METHOD M_Run
IF NOT _attached THEN
    RETURN;
END_IF
CASE _step OF
    0:  // initialize
        M_Step(StepNo := 0, StepName := 'project.step.pressAutoInitialize',
            Awaits := 0, AwaitingLabel := '', TimeClass := E_TimeClass.WORK, ExpectedTime := T#0S, Branch := 0);
        _outCmd.CycleCompleted := FALSE;
        _retVal := E_StepResult.ADVANCE;
        M_Advance(OnAdvance := 100, OnJump1 := -1, OnJump2 := -1, OnJump3 := -1 );
    100:  // await a fresh two-hand start (the §8.11.1 cycle-start marker)
        M_Step(StepNo := 100, StepName := 'project.step.pressAwaitTwoHand',
            Awaits := 0, AwaitingLabel := '', TimeClass := E_TimeClass.WAIT_OPERATOR, ExpectedTime := T#0S, Branch := 0);
        _outCmd.CycleCompleted := FALSE;
        _partReady := M_Await(Idx := 1, Label := 'project.condition.partPresent',
            Ok := _partPresentSensor.OutImm.Value AND _partPresentSensor.OutImm.Quality);
        _airReady := M_Await(Idx := 2, Label := 'project.condition.airPressureOk',
            Ok := _airPressureMonitor.OutImm.PressureOk);
        IF _stationCfg.RequireTwoHandStart THEN
            _startReady := M_Await(Idx := 3, Label := 'project.condition.twoHandStart', Ok := _startLatched);
        ELSE
            _startReady := TRUE;
        END_IF
        IF M_StopPending() THEN
            M_StopNow();                       // stop accepted BETWEEN cycles: no phantom cycle
        ELSIF _partReady AND _airReady AND _startReady THEN
            // §3.16.3 receive once per PHYSICAL part. The N180 two-hand abort returns
            // here with the same part still in the machine and nothing processed, so a
            // second M_PartReceived would open a duplicate record for one part.
            // M_PartStarted (N150) is deliberately NOT guarded: each pass is a genuine
            // processing attempt on that part.
            IF NOT _partInMachine THEN
                _traceAccepted := M_PartReceived();
                _partInMachine := TRUE;
            END_IF
            _retVal := E_StepResult.ADVANCE;
        END_IF
        M_Advance(OnAdvance := 110, OnJump1 := -1, OnJump2 := -1, OnJump3 := -1);
    110:  // ram up
        M_Step(StepNo := 110, StepName := 'project.step.pressRamUp',
            Awaits := _pressRam, AwaitingLabel := 'PressRam.RETRACT', TimeClass := E_TimeClass.WORK, ExpectedTime := T#0S, Branch := 0);
        IF M_TryIssue(Steppable := TRUE) THEN
            _pressRam.Abort := FALSE; _pressRam.Command := E_CylinderCommand.RETRACT; _pressRam.Execute := TRUE;
        END_IF
        IF _pressRam.Done THEN _pressRam.Execute := FALSE; _retVal := E_StepResult.ADVANCE; END_IF
        M_Advance(OnAdvance := 130, OnJump1 := -1, OnJump2 := -1, OnJump3 := -1);
    130:  // door open
        M_Step(StepNo := 130, StepName := 'project.step.pressDoorOpen',
            Awaits := _door, AwaitingLabel := 'Door.RETRACT', TimeClass := E_TimeClass.WORK, ExpectedTime := T#0S, Branch := 0);
        IF M_TryIssue(Steppable := TRUE) THEN
            _door.Abort := FALSE; _door.Command := E_CylinderCommand.RETRACT; _door.Execute := TRUE;
        END_IF
        IF _door.Done THEN _door.Execute := FALSE; _retVal := E_StepResult.ADVANCE; END_IF
        M_Advance(OnAdvance := 150, OnJump1 := -1, OnJump2 := -1, OnJump3 := -1);
    150:  // slide inside (value-adding sequence begins)
        M_Step(StepNo := 150, StepName := 'project.step.pressSlideInside',
            Awaits := _partSlide, AwaitingLabel := 'PartSlide.EXTEND', TimeClass := E_TimeClass.WORK, ExpectedTime := T#0S, Branch := 0);
        IF M_TryIssue(Steppable := TRUE) THEN
            M_PartStarted();
            _partSlide.Abort := FALSE; _partSlide.Command := E_CylinderCommand.EXTEND; _partSlide.Execute := TRUE;
        END_IF
        IF _partSlide.Done THEN _partSlide.Execute := FALSE; _retVal := E_StepResult.ADVANCE; END_IF
        M_Advance(OnAdvance := 170, OnJump1 := -1, OnJump2 := -1, OnJump3 := -1);
    170:  // transfer settle
        M_Step(StepNo := 170, StepName := 'project.step.pressTransferSettle',
            Awaits := 0, AwaitingLabel := '', TimeClass := E_TimeClass.WORK, ExpectedTime := _parCfg.TransferSettleTime, Branch := 0);
        _retVal := M_Delay(PT := _parCfg.TransferSettleTime);
        M_Advance(OnAdvance := 180, OnJump1 := -1, OnJump2 := -1, OnJump3 := -1);
    180:  // door close. Releasing a two-hand button while the door is moving is an
          // operator abort, not a fault: the door goes back up, the part slides out,
          // and the cycle returns to the two-hand wait (§6.10 jump). Completion wins
          // if the door finished in the same scan the button was released.
        M_Step(StepNo := 180, StepName := 'project.step.pressDoorClose',
            Awaits := _door, AwaitingLabel := 'Door.EXTEND', TimeClass := E_TimeClass.WORK, ExpectedTime := T#0S, Branch := 0);
        _twoHandHeldDuringClose := M_Await(Idx := 1,
            Label := 'project.condition.twoHandHeldDuringDoorClose',
            Ok := _twoHand.OutImm.SafeActive OR NOT _stationCfg.RequireTwoHandStart);
        IF M_TryIssue(Steppable := TRUE) THEN
            _door.Abort := FALSE; _door.Command := E_CylinderCommand.EXTEND; _door.Execute := TRUE;
        END_IF
        IF _door.Done THEN
            _door.Execute := FALSE;
            _retVal := E_StepResult.ADVANCE;
        ELSIF NOT _twoHandHeldDuringClose THEN
            _door.Execute := FALSE;             // §6.1 Execute-drop reset releases the close
            // §6.9(e) — a WARNING, not a fault: the release is designed operator
            // behaviour and the chain already owns the recovery below, so nothing
            // stops. It is recorded because a cycle was abandoned with the part
            // still in the machine, and the §3.13 chart marks this step for it.
            // The base raises it once per visit however many scans this runs.
            _closeAbortWarned := M_RaiseWarning(
                Reason := PL_PressReasons.PRESS_TWO_HAND_RELEASED,
                DescriptionKey := 'project.warning.twoHandReleasedDuringDoorClose',
                Severity := E_Severity.LOW, Category := E_Category.PROCESS);
            _retVal := E_StepResult.JUMP1;      // released -> reopen and clear the part
        END_IF
        M_Advance(OnAdvance := 200, OnJump1 := 185, OnJump2 := -1, OnJump3 := -1);
    185:  // two-hand released during closing: take the door back up
        M_Step(StepNo := 185, StepName := 'project.step.pressDoorReopen',
            Awaits := _door, AwaitingLabel := 'Door.RETRACT', TimeClass := E_TimeClass.WORK, ExpectedTime := T#0S, Branch := 0);
        IF M_TryIssue(Steppable := TRUE) THEN
            _door.Abort := FALSE; _door.Command := E_CylinderCommand.RETRACT; _door.Execute := TRUE;
        END_IF
        IF _door.Done THEN _door.Execute := FALSE; _retVal := E_StepResult.ADVANCE; END_IF
        M_Advance(OnAdvance := 190, OnJump1 := -1, OnJump2 := -1, OnJump3 := -1);
    190:  // slide the part back out, then return to the two-hand wait. The start latch
          // is dropped so the cycle cannot resume without a fresh two-hand press.
        M_Step(StepNo := 190, StepName := 'project.step.pressSlideOutsideAfterAbort',
            Awaits := _partSlide, AwaitingLabel := 'PartSlide.RETRACT', TimeClass := E_TimeClass.WORK, ExpectedTime := T#0S, Branch := 0);
        IF M_TryIssue(Steppable := TRUE) THEN
            _partSlide.Abort := FALSE; _partSlide.Command := E_CylinderCommand.RETRACT; _partSlide.Execute := TRUE;
        END_IF
        IF _partSlide.Done THEN
            _partSlide.Execute := FALSE;
            _startLatched := FALSE;
            _retVal := E_StepResult.ADVANCE;
        END_IF
        M_Advance(OnAdvance := 100, OnJump1 := -1, OnJump2 := -1, OnJump3 := -1);
    200:  // ram down. THIS step owns the not-reached disposition, so it does NOT hand
          // the ram to the §6.9 auto-rollup: an awaited child fault is adopted by the
          // Unit (ERROR, _step := 0) before _M_Dispatch runs, and the chain would stop
          // before it could ask the operator anything. The wait is still named (§6.9(b))
          // and the cylinder still raises its own CYL_NOT_EXTENDED alarm.
        M_Step(StepNo := 200, StepName := 'project.step.pressRamDown',
            Awaits := 0, AwaitingLabel := '', TimeClass := E_TimeClass.WORK, ExpectedTime := T#0S, Branch := 0);
        _ramReached := M_Await(Idx := 1, Label := 'project.condition.pressRamExtended',
            Ok := _pressRam.Done);
        IF M_TryIssue(Steppable := TRUE) THEN
            _pressRam.Abort := FALSE; _pressRam.Command := E_CylinderCommand.EXTEND; _pressRam.Execute := TRUE;
        END_IF
        IF _pressRam.Done THEN
            _pressRam.Execute := FALSE;
            _retVal := E_StepResult.ADVANCE;
        ELSIF _pressRam.Error THEN
            // §6.9(e) — publish the ram's own first-out (CYL_NOT_EXTENDED, with its
            // text and IO tag) on the Unit and on this row of the §3.13 chart, and
            // do NOT adopt it: the confirmation + scrap below IS the handling, so a
            // fault here would replace a designed recovery. Saying nothing is what
            // left the failure visible only on the ram itself.
            _ramFailureReported := M_ReportFromChild(Source := _pressRam);
            _pressRam.Execute := FALSE;         // §6.1 Execute-drop reset returns the ram to READY
            _retVal := E_StepResult.JUMP1;      // did not reach -> operator confirmation
        END_IF
        M_Advance(OnAdvance := 220, OnJump1 := 210, OnJump2 := -1, OnJump3 := -1);
    210:  // press did not reach: the operator confirms the failure before the part is
          // scrapped. A scrap is deliberate, so there is no timeout default (§6.11).
        M_Step(StepNo := 210, StepName := 'project.step.pressNotReachedConfirm',
            Awaits := 0, AwaitingLabel := '', TimeClass := E_TimeClass.WAIT_OPERATOR, ExpectedTime := T#0S, Branch := 0);
        _decisionRequest.Prompt := 'project.decision.pressNotReached';
        _decisionRequest.Options[1] := 'project.decision.confirmScrapAndReturn';
        _decisionRequest.Default := 0;
        _decisionRequest.Timeout := T#0S;
        M_AskDecision(Req := _decisionRequest);
        _answer := M_TakeDecision();
        IF _answer = 1 THEN
            _retVal := E_StepResult.ADVANCE;
        ELSE
            _failureConfirmed := M_Await(Idx := 1,
                Label := 'project.condition.pressFailureConfirmation', Ok := FALSE);
        END_IF
        M_Advance(OnAdvance := 215, OnJump1 := -1, OnJump2 := -1, OnJump3 := -1);
    215:  // disposition the part NOK, then rejoin the shared return-to-start step
        M_Step(StepNo := 215, StepName := 'project.step.pressScrapPart',
            Awaits := 0, AwaitingLabel := '', TimeClass := E_TimeClass.WORK, ExpectedTime := T#0S, Branch := 0);
        _partProcessed := M_PartProcessed(Verdict := E_Verdict.NOK,
            Reason := PL_ModuleReasons.CYL_NOT_EXTENDED);
        _partDispositioned := TRUE;             // N999 must not also count it good
        _partInMachine := FALSE;                // dispositioned: the next one is a new part
        _outCmd.CycleCompleted := FALSE;
        _retVal := E_StepResult.ADVANCE;
        M_Advance(OnAdvance := 240, OnJump1 := -1, OnJump2 := -1, OnJump3 := -1);
    220:  // press dwell — two-hand must stay held; releasing it HOLDS the dwell
        M_Step(StepNo := 220, StepName := 'project.step.pressDwell',
            Awaits := 0, AwaitingLabel := '', TimeClass := E_TimeClass.WORK, ExpectedTime := _parCfg.PressSettleTime, Branch := 0);
        // Releasing the button mid-dwell is the designed way to stop pressing, so it
        // is a named wait (§6.9(b)), not a fault: the ram's outputs come off, the
        // dwell timer freezes where it is because M_Delay is not called, and pressing
        // again restores the force and finishes the remaining dwell. Faulting here
        // charged an unrecoverable downtime event for normal operator behaviour.
        _dwellTwoHandHeld := M_Await(Idx := 1, Label := 'project.condition.twoHandHeldDuringPress',
            Ok := _twoHand.OutImm.SafeActive OR NOT _stationCfg.RequireTwoHandStart);
        IF NOT _dwellTwoHandHeld THEN
            _pressRam.WithdrawOutputs();
        ELSE
            // The press force is the valve latched by the EXTEND that step 200 already
            // completed, so after a withdraw only this call re-energizes it — and the
            // ram re-checks its own extend permit before it does (§7.2).
            _pressRam.RestoreOutputs();
            _retVal := M_Delay(PT := _parCfg.PressSettleTime);
        END_IF
        M_Advance(OnAdvance := 230, OnJump1 := -1, OnJump2 := -1, OnJump3 := -1);
    230:  // record the applied dwell (§3.16.1 measured value)
        M_Step(StepNo := 230, StepName := 'project.step.pressRecordResult',
            Awaits := 0, AwaitingLabel := '', TimeClass := E_TimeClass.WORK, ExpectedTime := T#0S, Branch := 0);
        _recordAccepted := M_PartRecord(RecordName := 'PressDwell',
            Value := DINT_TO_LREAL(TIME_TO_DINT(_parCfg.PressSettleTime)),
            Minimum := 0, Maximum := 30000,
            Target := DINT_TO_LREAL(TIME_TO_DINT(_parCfg.PressSettleTime)), EngUnit := 'ms');
        _retVal := E_StepResult.ADVANCE;
        M_Advance(OnAdvance := 240, OnJump1 := -1, OnJump2 := -1, OnJump3 := -1);
    240:  // return to the shared load-safe position (composite step)
        _retVal := M_RunSub(Chain := _loadPosition, BaseStepNo := 240);
        M_Advance(OnAdvance := 999, OnJump1 := -1, OnJump2 := -1, OnJump3 := -1);
    999:  // cycle complete — write result, count by verdict, loop (§8.11.1 finish marker)
        M_Step(StepNo := 999, StepName := 'project.step.pressAutoComplete',
            Awaits := 0, AwaitingLabel := '', TimeClass := E_TimeClass.WORK, ExpectedTime := T#0S, Branch := 0);
        _outCmd.CycleCompleted := TRUE;
        IF _partDispositioned THEN
            _partDispositioned := FALSE;       // N260 already set the NOK verdict
        ELSE
            _partProcessed := M_PartProcessed(Verdict := E_Verdict.OK, Reason := E_Reason.NONE);
            IF NOT _partProcessed THEN
                M_CountGood();                 // §3.9: no carrier configured — count directly
            END_IF
        END_IF
        _partInMachine := FALSE;               // processed: the next one is a new part
        _startLatched := FALSE;
        IF M_EndOfCycle() THEN
            _retVal := E_StepResult.ADVANCE;   // stop NOT requested: loop to N100
        END_IF
        M_Advance(OnAdvance := 100, OnJump1 := -1, OnJump2 := -1, OnJump3 := -1);
ELSE
    M_Fault(Reason := E_Reason.STEP_STALLED, DescriptionKey := 'std.error.undefinedStep');
END_CASE
END_METHOD

METHOD Setup : BOOL
VAR_INPUT
    Host : I_SequenceHost;
END_VAR
VAR_IN_OUT
    PressRam : FB_CylinderCM;
    Door : FB_CylinderCM;
    PartSlide : FB_CylinderCM;
    TwoHand : FB_TwoHandStartCM;
    PartPresentSensor : FB_DigitalInputCM;
    AirPressureMonitor : FB_AirPressureMonitorCM;
    ParCfg : ST_PneumaticPressParCfg;
    StationCfg : ST_PneumaticPressStationCfg;
    OutCmd : ST_PneumaticPressOutCmd;
    StartLatched : BOOL;
END_VAR
_pressRam REF= PressRam;
_door REF= Door;
_partSlide REF= PartSlide;
_twoHand REF= TwoHand;
_partPresentSensor REF= PartPresentSensor;
_airPressureMonitor REF= AirPressureMonitor;
_parCfg REF= ParCfg;
_stationCfg REF= StationCfg;
_outCmd REF= OutCmd;
_startLatched REF= StartLatched;
Setup := M_Attach(Host := Host) AND __ISVALIDREF(_pressRam) AND __ISVALIDREF(_door)
    AND __ISVALIDREF(_partSlide) AND __ISVALIDREF(_twoHand)
    AND __ISVALIDREF(_partPresentSensor) AND __ISVALIDREF(_airPressureMonitor)
    AND __ISVALIDREF(_parCfg) AND __ISVALIDREF(_outCmd) AND __ISVALIDREF(_startLatched)
    AND _loadPosition.Setup(Host := Host, PressRam := PressRam, Door := Door, PartSlide := PartSlide);
END_METHOD

END_FUNCTION_BLOCK

// ---- Fraktal_Press_Demo/01_PneumaticPress/Sequences/FB_SFC_PressDemoAuto.TcPOU
// SFC rendition of FB_PressDemoAuto - identical behaviour, chart-language
// transitions. Every step action below sets the shared `_retVal`; the chart's
// transitions read it, and the owner calls M_BeginScan() once per PLC cycle
// before executing this chart so the result cannot survive into the next scan
// (Core §6.8). The ST twin remains FB_PressDemoAuto; keep the two in step.
FUNCTION_BLOCK INTERNAL FB_SFC_PressDemoAuto EXTENDS FB_SequenceBase
VAR
    _partReady, _airReady, _startReady : BOOL;
    _dwellTwoHandHeld : BOOL;          // N220 named wait: two-hand held through the dwell
    _decisionRequest : ST_DecisionRequest;   // §6.11 not-reached confirmation
    _answer : INT;
    _ramReached, _failureConfirmed : BOOL;   // N200/N210 named waits
    _twoHandHeldDuringClose : BOOL;
    _closeAbortWarned : BOOL;                // N180 §6.9(e) message result
    _ramFailureReported : BOOL;              // N200 §6.9(e) message result          // N180 named wait
    _partInMachine : BOOL;                   // §3.16.3 the part is already received
    _partDispositioned : BOOL;               // N260 already set the verdict
    _traceAccepted, _recordAccepted, _partProcessed : BOOL;
    {attribute 'OPC.UA.DA' := '0'}
    _pressRam : REFERENCE TO FB_CylinderCM;
    {attribute 'OPC.UA.DA' := '0'}
    _door : REFERENCE TO FB_CylinderCM;
    {attribute 'OPC.UA.DA' := '0'}
    _partSlide : REFERENCE TO FB_CylinderCM;
    {attribute 'OPC.UA.DA' := '0'}
    _twoHand : REFERENCE TO FB_TwoHandStartCM;
    {attribute 'OPC.UA.DA' := '0'}
    _partPresentSensor : REFERENCE TO FB_DigitalInputCM;
    {attribute 'OPC.UA.DA' := '0'}
    _airPressureMonitor : REFERENCE TO FB_AirPressureMonitorCM;
    {attribute 'OPC.UA.DA' := '0'}
    _parCfg : REFERENCE TO ST_PneumaticPressParCfg;
    // §3.8a - the CELL's own policy, held separately from the MODEL's data and
    // referenced exactly like _parCfg, so each step reads whichever structure
    // actually owns the value it is asking about.
    {attribute 'OPC.UA.DA' := '0'}
    _stationCfg : REFERENCE TO ST_PneumaticPressStationCfg;
    {attribute 'OPC.UA.DA' := '0'}
    _outCmd : REFERENCE TO ST_PneumaticPressOutCmd;
    {attribute 'OPC.UA.DA' := '0'}
    _startLatched : REFERENCE TO BOOL;
    {attribute 'OPC.UA.DA' := '0'}
    _loadPosition : FB_PressDemoLoadPosition;
END_VAR

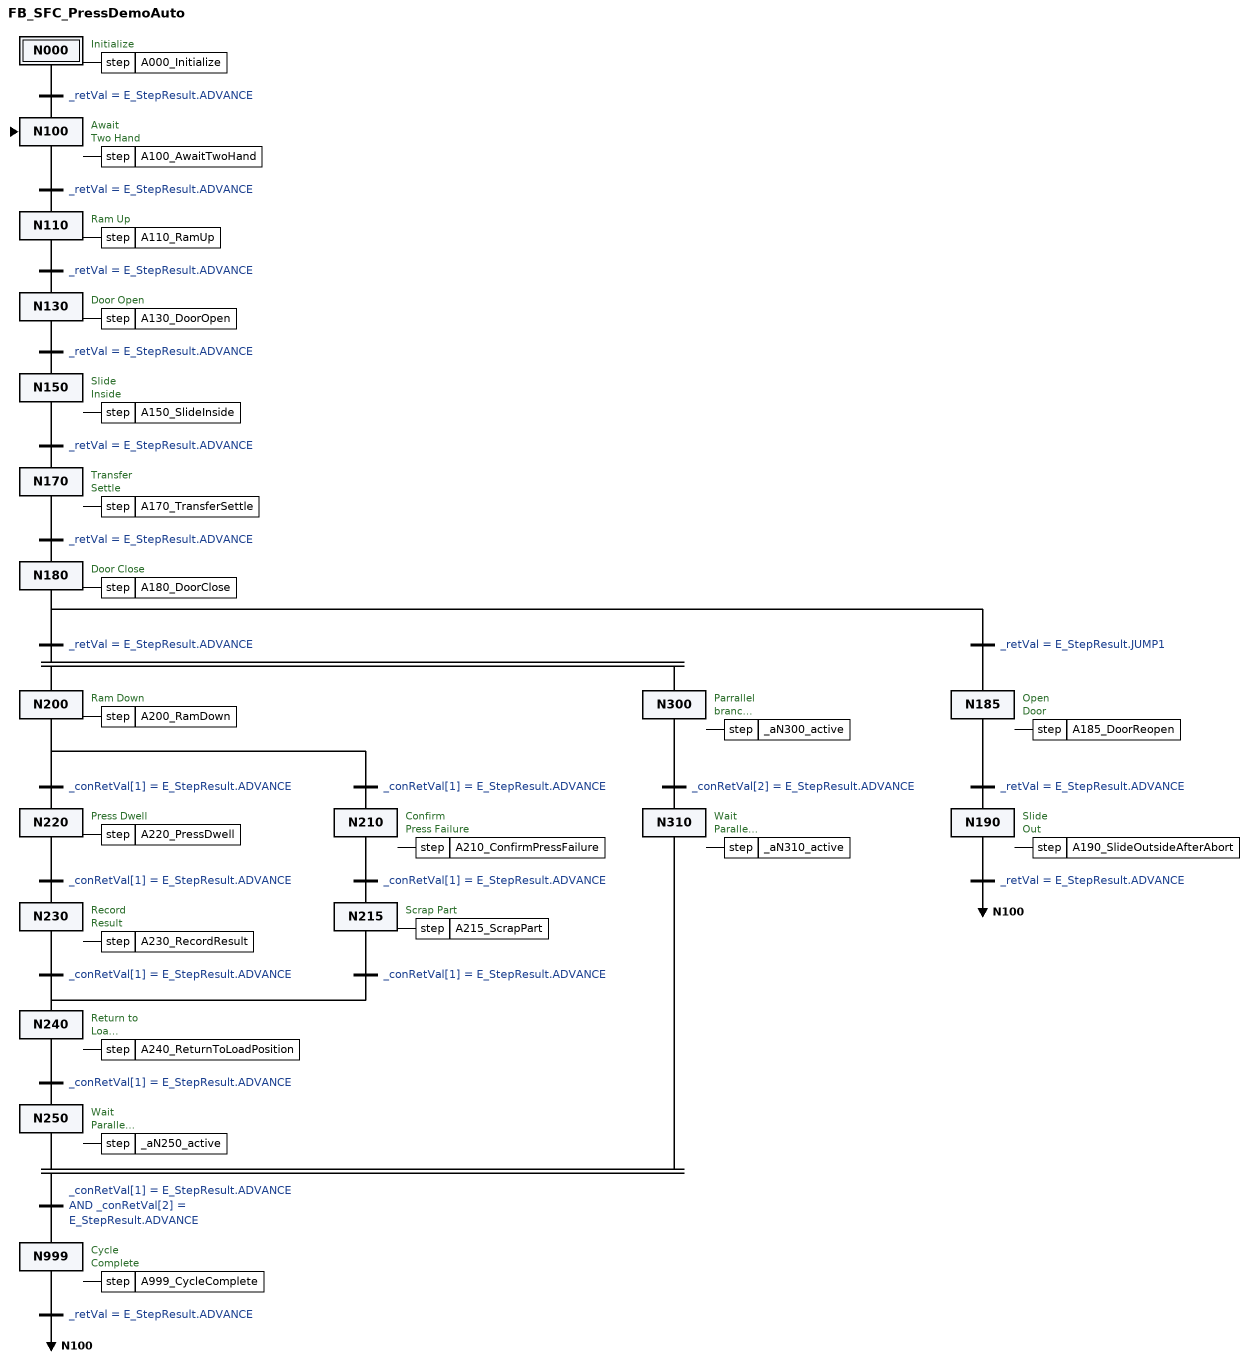
// Initialize
INITIAL_STEP N000:
    A000_Initialize(N);  // step action
END_STEP
TRANSITION FROM N000 TO N100
    := _retVal = E_StepResult.ADVANCE;
END_TRANSITION
// Await
// Two Hand
STEP N100:
    A100_AwaitTwoHand(N);  // step action
END_STEP
TRANSITION FROM N100 TO N110
    := _retVal = E_StepResult.ADVANCE;
END_TRANSITION
// Ram Up
STEP N110:
    A110_RamUp(N);  // step action
END_STEP
TRANSITION FROM N110 TO N130
    := _retVal = E_StepResult.ADVANCE;
END_TRANSITION
// Door Open
STEP N130:
    A130_DoorOpen(N);  // step action
END_STEP
TRANSITION FROM N130 TO N150
    := _retVal = E_StepResult.ADVANCE;
END_TRANSITION
// Slide
// Inside
STEP N150:
    A150_SlideInside(N);  // step action
END_STEP
TRANSITION FROM N150 TO N170
    := _retVal = E_StepResult.ADVANCE;
END_TRANSITION
// Transfer
// Settle
STEP N170:
    A170_TransferSettle(N);  // step action
END_STEP
TRANSITION FROM N170 TO N180
    := _retVal = E_StepResult.ADVANCE;
END_TRANSITION
// Door Close
STEP N180:
    A180_DoorClose(N);  // step action
END_STEP
TRANSITION FROM N180 TO (N200, N300)
    := _retVal = E_StepResult.ADVANCE;
END_TRANSITION
// Ram Down
STEP N200:
    A200_RamDown(N);  // step action
END_STEP
TRANSITION FROM N200 TO N220
    := _conRetVal[1] = E_StepResult.ADVANCE;
END_TRANSITION
// Press Dwell
STEP N220:
    A220_PressDwell(N);  // step action
END_STEP
TRANSITION FROM N220 TO N230
    := _conRetVal[1] = E_StepResult.ADVANCE;
END_TRANSITION
// Record
// Result
STEP N230:
    A230_RecordResult(N);  // step action
END_STEP
TRANSITION FROM N230 TO N240
    := _conRetVal[1] = E_StepResult.ADVANCE;
END_TRANSITION
TRANSITION FROM N200 TO N210
    := _conRetVal[1] = E_StepResult.ADVANCE;
END_TRANSITION
// Confirm
// Press Failure
STEP N210:
    A210_ConfirmPressFailure(N);  // step action
END_STEP
TRANSITION FROM N210 TO N215
    := _conRetVal[1] = E_StepResult.ADVANCE;
END_TRANSITION
// Scrap Part
STEP N215:
    A215_ScrapPart(N);  // step action
END_STEP
TRANSITION FROM N215 TO N240
    := _conRetVal[1] = E_StepResult.ADVANCE;
END_TRANSITION
// Return to
// Load
// Position
STEP N240:
    A240_ReturnToLoadPosition(N);  // step action
END_STEP
TRANSITION FROM N240 TO N250
    := _conRetVal[1] = E_StepResult.ADVANCE;
END_TRANSITION
// Wait
// Parallel
// Branch
STEP N250:
    _aN250_active(N);  // step action
END_STEP
// Parrallel
// branch
// example
STEP N300:
    _aN300_active(N);  // step action
END_STEP
TRANSITION FROM N300 TO N310
    := _conRetVal[2] = E_StepResult.ADVANCE;
END_TRANSITION
// Wait
// Parallel
// Branch
STEP N310:
    _aN310_active(N);  // step action
END_STEP
TRANSITION FROM N180 TO N185
    := _retVal = E_StepResult.JUMP1;
END_TRANSITION
// Open
// Door
STEP N185:
    A185_DoorReopen(N);  // step action
END_STEP
TRANSITION FROM N185 TO N190
    := _retVal = E_StepResult.ADVANCE;
END_TRANSITION
// Slide
// Out
STEP N190:
    A190_SlideOutsideAfterAbort(N);  // step action
END_STEP
TRANSITION FROM N190 TO N100
    := _retVal = E_StepResult.ADVANCE;
END_TRANSITION
TRANSITION FROM (N250, N310) TO N999
    := _conRetVal[1] = E_StepResult.ADVANCE AND _conRetVal[2] = E_StepResult.ADVANCE;
END_TRANSITION
// Cycle
// Complete
STEP N999:
    A999_CycleComplete(N);  // step action
END_STEP
TRANSITION FROM N999 TO N100
    := _retVal = E_StepResult.ADVANCE;
END_TRANSITION

ACTION _aN250_active:
// N250 — leg 1 waits at the join. §6.12: the parallel divergence after A180 is
// drawn INSIDE this POU, so both legs share the FB and each leg step says which leg
// it is through `Branch` on its own step record - a leg can never be declared
// without recording a step.
//
// NEITHER leg is the main line. A simultaneous divergence has N equal legs, so
// numbering one of them 0 would have made it look subordinate on the §3.13 chart
// and left `_retVal` meaning two different things depending on where you were
// reading it. `_retVal` is the single-threaded line before and after the fork;
// inside it, leg 1 is `_conRetVal[1]` and leg 2 is `_conRetVal[2]`.
M_Step(StepNo := 250, StepName := 'project.step.pressAwaitParallelBranch', Awaits := 0,
    AwaitingLabel := '', TimeClass := E_TimeClass.WORK, ExpectedTime := T#0S,
    Branch := 1);
_conRetVal[1] := E_StepResult.ADVANCE;
END_ACTION

ACTION _aN300_active:
// N300 — concurrent leg 1, first step. Everything a normal step does is available
// here; `Branch := 1` is what keeps this leg's issue latch, delay and message
// separate from the main line's, so both legs can command their own children in
// the same scan. This example commands nothing: the press has one work position,
// and inventing a second would change what the machine does. A real one goes here.
M_Step(StepNo := 300, StepName := 'project.step.pressParallelWork', Awaits := 0,
    AwaitingLabel := '', TimeClass := E_TimeClass.WORK, ExpectedTime := T#0S,
    Branch := 2);
_conRetVal[2] := E_StepResult.ADVANCE;   // leg 2's result; leg 1 uses _conRetVal[1]
END_ACTION

ACTION _aN310_active:
// N310 — concurrent leg 1 waits at the join. A parallel divergence joins only when
// EVERY leg has reached its last step, so each leg needs a terminal step to sit in
// while the others finish; this is that step for leg 1, and A250 is the main
// line's.
M_Step(StepNo := 310, StepName := 'project.step.pressAwaitParallelJoin', Awaits := 0,
    AwaitingLabel := '', TimeClass := E_TimeClass.WORK, ExpectedTime := T#0S,
    Branch := 2);
_conRetVal[2] := E_StepResult.ADVANCE;
END_ACTION

ACTION A000_Initialize:
// N000 step action. SFC step `A000_Initialize` calls this; its transition reads
// `_retVal = E_StepResult.ADVANCE`. Body is the ST chart's branch verbatim,
// without M_Advance - the chart runtime owns the transition.
M_Step(StepNo := 0, StepName := 'project.step.pressAutoInitialize',
    Awaits := 0, AwaitingLabel := '', TimeClass := E_TimeClass.WORK, ExpectedTime := T#0S, Branch := 0);
_outCmd.CycleCompleted := FALSE;
_retVal := E_StepResult.ADVANCE;
END_ACTION

ACTION A100_AwaitTwoHand:
// N100 step action. The §8.11.1 cycle-start marker; also the target of the
// N190 two-hand abort, which returns here with the same part still in place.
M_Step(StepNo := 100, StepName := 'project.step.pressAwaitTwoHand',
    Awaits := 0, AwaitingLabel := '', TimeClass := E_TimeClass.WAIT_OPERATOR, ExpectedTime := T#0S, Branch := 0);
_outCmd.CycleCompleted := FALSE;
_partReady := M_Await(Idx := 1, Label := 'project.condition.partPresent',
    Ok := _partPresentSensor.OutImm.Value AND _partPresentSensor.OutImm.Quality);
_airReady := M_Await(Idx := 2, Label := 'project.condition.airPressureOk',
    Ok := _airPressureMonitor.OutImm.PressureOk);
IF _stationCfg.RequireTwoHandStart THEN
    _startReady := M_Await(Idx := 3, Label := 'project.condition.twoHandStart', Ok := _startLatched);
ELSE
    _startReady := TRUE;
END_IF
IF M_StopPending() THEN
    M_StopNow();                       // stop accepted BETWEEN cycles: no phantom cycle
ELSIF _partReady AND _airReady AND _startReady THEN
    // §3.16.3 receive once per PHYSICAL part. The N180 two-hand abort returns
    // here with the same part still in the machine and nothing processed, so a
    // second M_PartReceived would open a duplicate record for one part.
    // M_PartStarted (N150) is deliberately NOT guarded: each pass is a genuine
    // processing attempt on that part.
    IF NOT _partInMachine THEN
        _traceAccepted := M_PartReceived();
        _partInMachine := TRUE;
    END_IF
    _retVal := E_StepResult.ADVANCE;
END_IF
END_ACTION

ACTION A110_RamUp:
// N110 step action. SFC step `A110_RamUp` calls this; its transition reads
// `_retVal = E_StepResult.ADVANCE`. Body is the ST chart's branch verbatim,
// without M_Advance - the chart runtime owns the transition.
M_Step(StepNo := 110, StepName := 'project.step.pressRamUp',
    Awaits := _pressRam, AwaitingLabel := 'PressRam.RETRACT', TimeClass := E_TimeClass.WORK, ExpectedTime := T#0S, Branch := 0);
IF M_TryIssue(Steppable := TRUE) THEN
    _pressRam.Abort := FALSE; _pressRam.Command := E_CylinderCommand.RETRACT; _pressRam.Execute := TRUE;
END_IF
IF _pressRam.Done THEN _pressRam.Execute := FALSE; _retVal := E_StepResult.ADVANCE; END_IF
END_ACTION

ACTION A130_DoorOpen:
// N130 step action. SFC step `A130_DoorOpen` calls this; its transition reads
// `_retVal = E_StepResult.ADVANCE`. Body is the ST chart's branch verbatim,
// without M_Advance - the chart runtime owns the transition.
M_Step(StepNo := 130, StepName := 'project.step.pressDoorOpen',
    Awaits := _door, AwaitingLabel := 'Door.RETRACT', TimeClass := E_TimeClass.WORK, ExpectedTime := T#0S, Branch := 0);
IF M_TryIssue(Steppable := TRUE) THEN
    _door.Abort := FALSE; _door.Command := E_CylinderCommand.RETRACT; _door.Execute := TRUE;
END_IF
IF _door.Done THEN _door.Execute := FALSE; _retVal := E_StepResult.ADVANCE; END_IF
END_ACTION

ACTION A150_SlideInside:
// N150 step action. SFC step `A150_SlideInside` calls this; its transition reads
// `_retVal = E_StepResult.ADVANCE`. Body is the ST chart's branch verbatim,
// without M_Advance - the chart runtime owns the transition.
M_Step(StepNo := 150, StepName := 'project.step.pressSlideInside',
    Awaits := _partSlide, AwaitingLabel := 'PartSlide.EXTEND', TimeClass := E_TimeClass.WORK, ExpectedTime := T#0S, Branch := 0);
IF M_TryIssue(Steppable := TRUE) THEN
    M_PartStarted();
    _partSlide.Abort := FALSE; _partSlide.Command := E_CylinderCommand.EXTEND; _partSlide.Execute := TRUE;
END_IF
IF _partSlide.Done THEN _partSlide.Execute := FALSE; _retVal := E_StepResult.ADVANCE; END_IF
END_ACTION

ACTION A170_TransferSettle:
// N170 step action. SFC step `A170_TransferSettle` calls this; its transition reads
// `_retVal = E_StepResult.ADVANCE`. Body is the ST chart's branch verbatim,
// without M_Advance - the chart runtime owns the transition.
M_Step(StepNo := 170, StepName := 'project.step.pressTransferSettle',
    Awaits := 0, AwaitingLabel := '', TimeClass := E_TimeClass.WORK, ExpectedTime := _parCfg.TransferSettleTime, Branch := 0);
_retVal := M_Delay(PT := _parCfg.TransferSettleTime);
END_ACTION

ACTION A180_DoorClose:
// N180 step action. Transition `_retVal = E_StepResult.ADVANCE` -> A200;
// the JUMP1 branch (`_retVal = E_StepResult.JUMP1`) -> A185.
//
// Releasing a two-hand button while the door is moving is an operator abort, not
// a fault: the door goes back up, the part slides out, and the cycle returns to
// the two-hand wait. Completion wins if the door finished in the same scan the
// button was released.
M_Step(StepNo := 180, StepName := 'project.step.pressDoorClose',
    Awaits := _door, AwaitingLabel := 'Door.EXTEND', TimeClass := E_TimeClass.WORK, ExpectedTime := T#0S, Branch := 0);
_twoHandHeldDuringClose := M_Await(Idx := 1,
    Label := 'project.condition.twoHandHeldDuringDoorClose',
    Ok := _twoHand.OutImm.SafeActive OR NOT _stationCfg.RequireTwoHandStart);
IF M_TryIssue(Steppable := TRUE) THEN
    _door.Abort := FALSE; _door.Command := E_CylinderCommand.EXTEND; _door.Execute := TRUE;
END_IF
IF _door.Done THEN
    _door.Execute := FALSE;
    _retVal := E_StepResult.ADVANCE;
ELSIF NOT _twoHandHeldDuringClose THEN
    _door.Execute := FALSE;             // §6.1 Execute-drop reset releases the close
    // §6.9(e) — a WARNING, not a fault: nothing stops, the JUMP1 branch below is
    // the recovery. Recorded because a cycle was abandoned with the part still in
    // the machine. Raised once per visit however many scans this action runs.
    _closeAbortWarned := M_RaiseWarning(
        Reason := PL_PressReasons.PRESS_TWO_HAND_RELEASED,
        DescriptionKey := 'project.warning.twoHandReleasedDuringDoorClose',
        Severity := E_Severity.LOW, Category := E_Category.PROCESS);
    _retVal := E_StepResult.JUMP1;      // released -> reopen and clear the part
END_IF
END_ACTION

ACTION A185_DoorReopen:
// N185 step action. Reached from A180 by JUMP1 when a two-hand button is
// released while the door closes. Advances to A190.
M_Step(StepNo := 185, StepName := 'project.step.pressDoorReopen',
    Awaits := _door, AwaitingLabel := 'Door.RETRACT', TimeClass := E_TimeClass.WORK, ExpectedTime := T#0S, Branch := 0);
IF M_TryIssue(Steppable := TRUE) THEN
    _door.Abort := FALSE; _door.Command := E_CylinderCommand.RETRACT; _door.Execute := TRUE;
END_IF
IF _door.Done THEN _door.Execute := FALSE; _retVal := E_StepResult.ADVANCE; END_IF
END_ACTION

ACTION A190_SlideOutsideAfterAbort:
// N190 step action. Slides the part out and drops the start latch, then its
// transition jumps back to A100, the two-hand wait. The start latch is dropped
// so the cycle cannot resume without a fresh two-hand press.
M_Step(StepNo := 190, StepName := 'project.step.pressSlideOutsideAfterAbort',
    Awaits := _partSlide, AwaitingLabel := 'PartSlide.RETRACT', TimeClass := E_TimeClass.WORK, ExpectedTime := T#0S, Branch := 0);
IF M_TryIssue(Steppable := TRUE) THEN
    _partSlide.Abort := FALSE; _partSlide.Command := E_CylinderCommand.RETRACT; _partSlide.Execute := TRUE;
END_IF
IF _partSlide.Done THEN
    _partSlide.Execute := FALSE;
    _startLatched := FALSE;
    _retVal := E_StepResult.ADVANCE;
END_IF
END_ACTION

ACTION A200_RamDown:
// N200 step action. Transition `_retVal = E_StepResult.ADVANCE` -> A220;
// the JUMP1 branch (`_retVal = E_StepResult.JUMP1`) -> A210.
// the ram to the §6.9 auto-rollup: an awaited child fault is adopted by the
// Unit (ERROR, _step := 0) before _M_Dispatch runs, and the chain would stop
// before it could ask the operator anything. The wait is still named (§6.9(b))
// and the cylinder still raises its own CYL_NOT_EXTENDED alarm.
M_Step(StepNo := 200, StepName := 'project.step.pressRamDown',
    Awaits := 0, AwaitingLabel := '', TimeClass := E_TimeClass.WORK, ExpectedTime := T#0S,
    Branch := 1);
_ramReached := M_Await(Idx := 1, Label := 'project.condition.pressRamExtended',
    Ok := _pressRam.Done);
IF M_TryIssue(Steppable := TRUE) THEN
    _pressRam.Abort := FALSE; _pressRam.Command := E_CylinderCommand.EXTEND; _pressRam.Execute := TRUE;
END_IF
IF _pressRam.Done THEN
    _pressRam.Execute := FALSE;
    _conRetVal[1] := E_StepResult.ADVANCE;
ELSIF _pressRam.Error THEN
    // §6.9(e) — publish the ram's own first-out on the Unit and on this row of the
    // §3.13 chart without adopting it: the confirmation + scrap below IS the
    // handling, so a fault here would replace a designed recovery.
    _ramFailureReported := M_ReportFromChild(Source := _pressRam);
    _pressRam.Execute := FALSE;         // §6.1 Execute-drop reset returns the ram to READY
    _conRetVal[1] := E_StepResult.JUMP1;      // did not reach -> operator confirmation
END_IF
END_ACTION

ACTION A210_ConfirmPressFailure:
// N210 step action. Reached from A200 by JUMP1; advances to A215.
// scrapped. A scrap is deliberate, so there is no timeout default (§6.11).
M_Step(StepNo := 210, StepName := 'project.step.pressNotReachedConfirm',
    Awaits := 0, AwaitingLabel := '', TimeClass := E_TimeClass.WAIT_OPERATOR, ExpectedTime := T#0S,
    Branch := 1);
_decisionRequest.Prompt := 'project.decision.pressNotReached';
_decisionRequest.Options[1] := 'project.decision.confirmScrapAndReturn';
_decisionRequest.Default := 0;
_decisionRequest.Timeout := T#0S;
M_AskDecision(Req := _decisionRequest);
_answer := M_TakeDecision();
IF _answer = 1 THEN
    _conRetVal[1] := E_StepResult.ADVANCE;
ELSE
    _failureConfirmed := M_Await(Idx := 1,
        Label := 'project.condition.pressFailureConfirmation', Ok := FALSE);
END_IF
END_ACTION

ACTION A215_ScrapPart:
// N215 step action. Sets the part NOK and releases it, then rejoins A240.
M_Step(StepNo := 215, StepName := 'project.step.pressScrapPart',
    Awaits := 0, AwaitingLabel := '', TimeClass := E_TimeClass.WORK, ExpectedTime := T#0S,
    Branch := 1);
_partProcessed := M_PartProcessed(Verdict := E_Verdict.NOK,
    Reason := PL_ModuleReasons.CYL_NOT_EXTENDED);
_partDispositioned := TRUE;             // N999 must not also count it good
_partInMachine := FALSE;                // dispositioned: the next one is a new part
_outCmd.CycleCompleted := FALSE;
_conRetVal[1] := E_StepResult.ADVANCE;
END_ACTION

ACTION A220_PressDwell:
// N220 step action. SFC step `A220_PressDwell` calls this; its transition reads
// `_retVal = E_StepResult.ADVANCE`. Body is the ST chart's branch verbatim,
// without M_Advance - the chart runtime owns the transition.
M_Step(StepNo := 220, StepName := 'project.step.pressDwell',
    Awaits := 0, AwaitingLabel := '', TimeClass := E_TimeClass.WORK, ExpectedTime := _parCfg.PressSettleTime,
    Branch := 1);
// Releasing the button mid-dwell is the designed way to stop pressing, so it
// is a named wait (§6.9(b)), not a fault: the ram's outputs come off, the
// dwell timer freezes where it is because M_Delay is not called, and pressing
// again restores the force and finishes the remaining dwell. Faulting here
// charged an unrecoverable downtime event for normal operator behaviour.
_dwellTwoHandHeld := M_Await(Idx := 1, Label := 'project.condition.twoHandHeldDuringPress',
    Ok := _twoHand.OutImm.SafeActive OR NOT _stationCfg.RequireTwoHandStart);
IF NOT _dwellTwoHandHeld THEN
    _pressRam.WithdrawOutputs();
ELSE
    // The press force is the valve latched by the EXTEND that step 200 already
    // completed, so after a withdraw only this call re-energizes it — and the
    // ram re-checks its own extend permit before it does (§7.2).
    _pressRam.RestoreOutputs();
    _conRetVal[1] := M_Delay(PT := _parCfg.PressSettleTime);
END_IF
END_ACTION

ACTION A230_RecordResult:
// N230 step action. SFC step `A230_RecordResult` calls this; its transition reads
// `_retVal = E_StepResult.ADVANCE`. Body is the ST chart's branch verbatim,
// without M_Advance - the chart runtime owns the transition.
M_Step(StepNo := 230, StepName := 'project.step.pressRecordResult',
    Awaits := 0, AwaitingLabel := '', TimeClass := E_TimeClass.WORK, ExpectedTime := T#0S,
    Branch := 1);
_recordAccepted := M_PartRecord(RecordName := 'PressDwell',
    Value := DINT_TO_LREAL(TIME_TO_DINT(_parCfg.PressSettleTime)),
    Minimum := 0, Maximum := 30000,
    Target := DINT_TO_LREAL(TIME_TO_DINT(_parCfg.PressSettleTime)), EngUnit := 'ms');
_conRetVal[1] := E_StepResult.ADVANCE;
END_ACTION

ACTION A240_ReturnToLoadPosition:
// N240 step action, on concurrent leg 1. Its transition reads
// `_conRetVal[1] = E_StepResult.ADVANCE`. Body is the ST chart's branch verbatim,
// without M_Advance - the chart runtime owns the transition.
//
// The sub-chain needs no leg argument: M_RunSub inherits the leg of the step that
// runs it (§6.12), so the load-position steps publish as leg 1 too.
_conRetVal[1] := M_RunSub(Chain := _loadPosition, BaseStepNo := 240);
END_ACTION

ACTION A999_CycleComplete:
// N999 step action. Transition `_retVal = E_StepResult.ADVANCE` loops to A100.
M_Step(StepNo := 999, StepName := 'project.step.pressAutoComplete',
    Awaits := 0, AwaitingLabel := '', TimeClass := E_TimeClass.WORK, ExpectedTime := T#0S, Branch := 0);
_outCmd.CycleCompleted := TRUE;
IF _partDispositioned THEN
    _partDispositioned := FALSE;       // N260 already set the NOK verdict
ELSE
    _partProcessed := M_PartProcessed(Verdict := E_Verdict.OK, Reason := E_Reason.NONE);
    IF NOT _partProcessed THEN
        M_CountGood();                 // §3.9: no carrier configured — count directly
    END_IF
END_IF
_partInMachine := FALSE;               // processed: the next one is a new part
_startLatched := FALSE;
IF M_EndOfCycle() THEN
    _retVal := E_StepResult.ADVANCE;   // stop NOT requested: loop to N100
END_IF
END_ACTION

// §6.8 - the chain's own state on a restart (the base resets the flow state).
METHOD PROTECTED OnChainReset
// A chart restart abandons whatever the cycle was holding: the part record is
// closed by N215/N999, never by a restart, so both trackers start clean.
_partDispositioned := FALSE;
_partInMachine := FALSE;
END_METHOD

METHOD Setup : BOOL
VAR_INPUT
    Host : I_SequenceHost;
END_VAR
VAR_IN_OUT
    PressRam : FB_CylinderCM;
    Door : FB_CylinderCM;
    PartSlide : FB_CylinderCM;
    TwoHand : FB_TwoHandStartCM;
    PartPresentSensor : FB_DigitalInputCM;
    AirPressureMonitor : FB_AirPressureMonitorCM;
    ParCfg : ST_PneumaticPressParCfg;
    StationCfg : ST_PneumaticPressStationCfg;
    OutCmd : ST_PneumaticPressOutCmd;
    StartLatched : BOOL;
END_VAR
_pressRam REF= PressRam;
_door REF= Door;
_partSlide REF= PartSlide;
_twoHand REF= TwoHand;
_partPresentSensor REF= PartPresentSensor;
_airPressureMonitor REF= AirPressureMonitor;
_parCfg REF= ParCfg;
_stationCfg REF= StationCfg;
_outCmd REF= OutCmd;
_startLatched REF= StartLatched;
Setup := M_Attach(Host := Host) AND __ISVALIDREF(_pressRam) AND __ISVALIDREF(_door)
    AND __ISVALIDREF(_partSlide) AND __ISVALIDREF(_twoHand)
    AND __ISVALIDREF(_partPresentSensor) AND __ISVALIDREF(_airPressureMonitor)
    AND __ISVALIDREF(_parCfg) AND __ISVALIDREF(_outCmd) AND __ISVALIDREF(_startLatched)
    AND _loadPosition.Setup(Host := Host, PressRam := PressRam, Door := Door, PartSlide := PartSlide);
END_METHOD

END_FUNCTION_BLOCK

// ---- Fraktal_Press_Demo/01_PneumaticPress/Sequences/FB_LD_PressDemoAuto.TcPOU
FUNCTION_BLOCK FB_LD_PressDemoAuto EXTENDS FB_SequenceBase
VAR
    _partReady, _airReady, _startReady, _stop, _doStep, _processed, _endCycle, _dummy : BOOL;
    _dwellTwoHandHeld : BOOL;          // N220 named wait: two-hand held through the dwell
    _decisionRequest : ST_DecisionRequest;   // §6.11 not-reached confirmation
    _answer : INT;
    _ramReached, _failureConfirmed : BOOL;   // N200/N210 named waits
    _twoHandHeldDuringClose : BOOL;          // N180 named wait
    _closeAbortWarned : BOOL;                // N180 §6.9(e) message result
    _ramFailureReported : BOOL;              // N200 §6.9(e) message result
    _partInMachine : BOOL;                   // §3.16.3 the part is already received
    _partDispositioned : BOOL;               // N260 already set the verdict
    _traceAccepted, _recordAccepted, _partProcessed : BOOL;
    {attribute 'OPC.UA.DA' := '0'}
    _pressRam : REFERENCE TO FB_CylinderCM;
    {attribute 'OPC.UA.DA' := '0'}
    _door : REFERENCE TO FB_CylinderCM;
    {attribute 'OPC.UA.DA' := '0'}
    _partSlide : REFERENCE TO FB_CylinderCM;
    {attribute 'OPC.UA.DA' := '0'}
    _twoHand : REFERENCE TO FB_TwoHandStartCM;
    {attribute 'OPC.UA.DA' := '0'}
    _partPresentSensor : REFERENCE TO FB_DigitalInputCM;
    {attribute 'OPC.UA.DA' := '0'}
    _airPressureMonitor : REFERENCE TO FB_AirPressureMonitorCM;
    {attribute 'OPC.UA.DA' := '0'}
    _parCfg : REFERENCE TO ST_PneumaticPressParCfg;
    // §3.8a - the cell's own policy, referenced like _parCfg.
    {attribute 'OPC.UA.DA' := '0'}
    _stationCfg : REFERENCE TO ST_PneumaticPressStationCfg;
    {attribute 'OPC.UA.DA' := '0'}
    _outCmd : REFERENCE TO ST_PneumaticPressOutCmd;
    {attribute 'OPC.UA.DA' := '0'}
    _startLatched : REFERENCE TO BOOL;
    {attribute 'OPC.UA.DA' := '0'}
    _loadPosition : FB_PressDemoLoadPosition;
END_VAR
VAR // added by the converter: edge detectors and wires of the graphical bodies
    _w1, _w2, _w3, _w4, _w5, _w6, _w7, _w8, _w9, _w10, _w11, _w12, _w13, _w14, _w15, _w16, _w17, _w18, _w19, _w20, _w21, _w22, _w23, _w24, _w25, _w26, _w27, _w28, _w29, _w30 : BOOL;
END_VAR

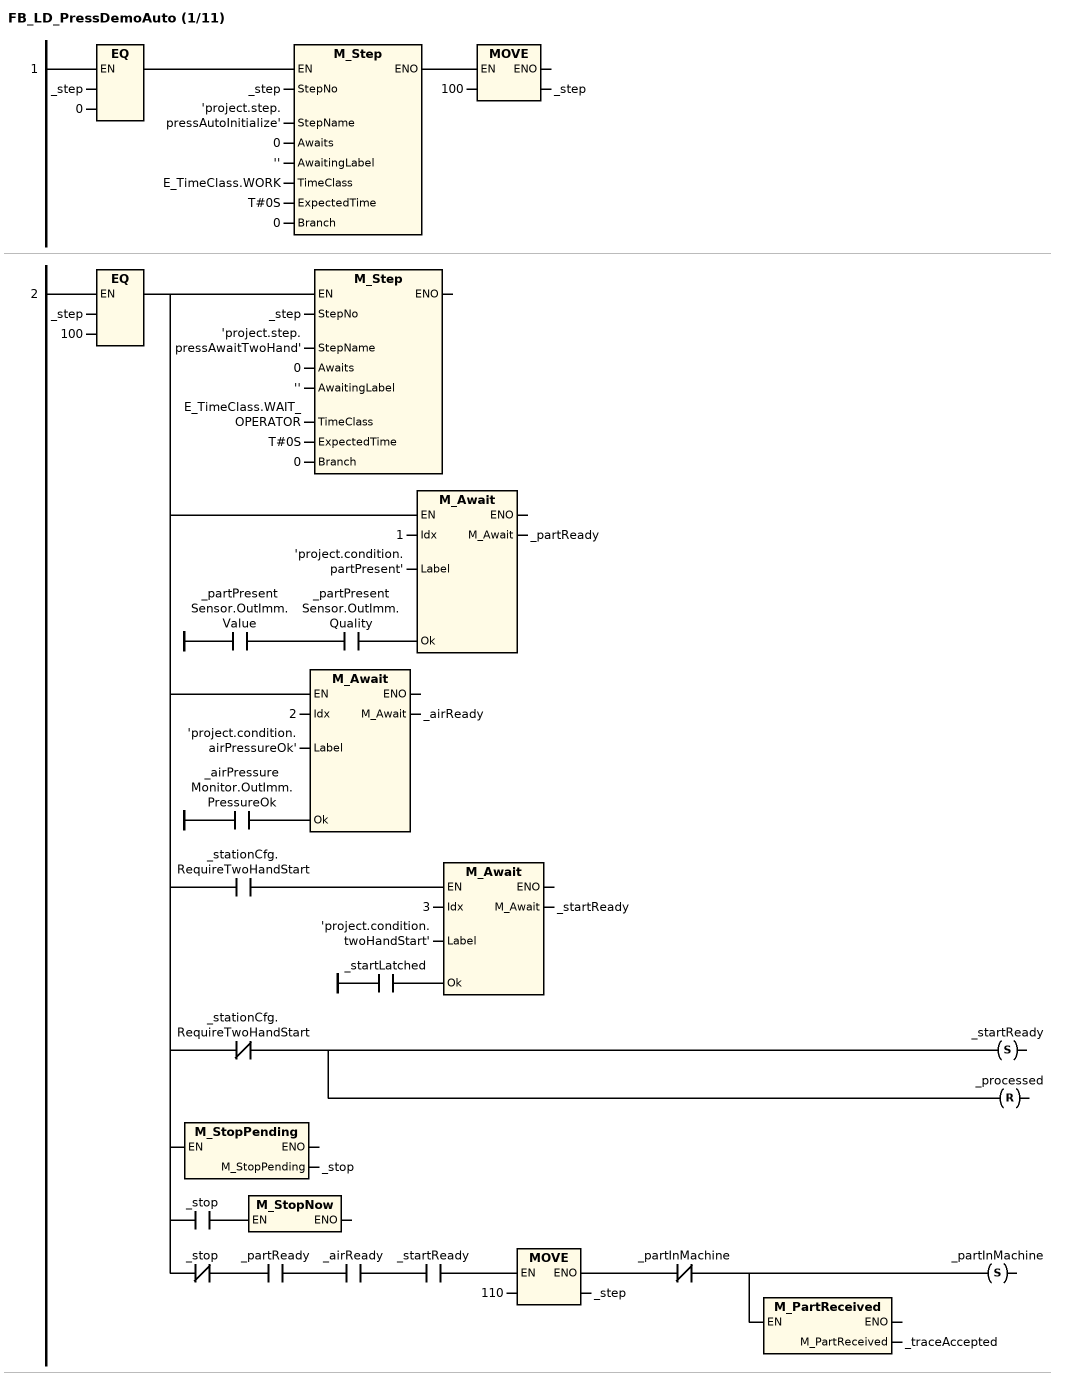
// NETWORK 1
_w1 := _step = 0;
IF _w1 THEN
    M_Step(StepNo := _step, StepName := 'project.step.pressAutoInitialize', Awaits := 0, AwaitingLabel := '', TimeClass := E_TimeClass.WORK, ExpectedTime := T#0S, Branch := 0);
END_IF
IF _w1 THEN _step := 100; END_IF

// NETWORK 2
_w2 := _step = 100;
IF _w2 THEN
    M_Step(StepNo := _step, StepName := 'project.step.pressAwaitTwoHand', Awaits := 0, AwaitingLabel := '', TimeClass := E_TimeClass.WAIT_OPERATOR, ExpectedTime := T#0S, Branch := 0);
END_IF
IF _w2 THEN
    _partReady := M_Await(Idx := 1, Label := 'project.condition.partPresent', Ok := _partPresentSensor.OutImm.Value AND _partPresentSensor.OutImm.Quality);
END_IF
IF _w2 THEN
    _airReady := M_Await(Idx := 2, Label := 'project.condition.airPressureOk', Ok := _airPressureMonitor.OutImm.PressureOk);
END_IF
IF _w2 AND _stationCfg.RequireTwoHandStart THEN
    _startReady := M_Await(Idx := 3, Label := 'project.condition.twoHandStart', Ok := _startLatched);
END_IF
_w3 := _w2 AND NOT _stationCfg.RequireTwoHandStart;
_startReady S= _w3;
_processed R= _w3;
IF _w2 THEN _stop := M_StopPending(); END_IF
IF _w2 AND _stop THEN M_StopNow(); END_IF
IF _w2 AND NOT _stop AND _partReady AND _airReady AND _startReady THEN _step := 110; END_IF
_w4 := (_w2 AND NOT _stop AND _partReady AND _airReady AND _startReady) AND NOT _partInMachine;
_partInMachine S= _w4;
IF _w4 THEN _traceAccepted := M_PartReceived(); END_IF

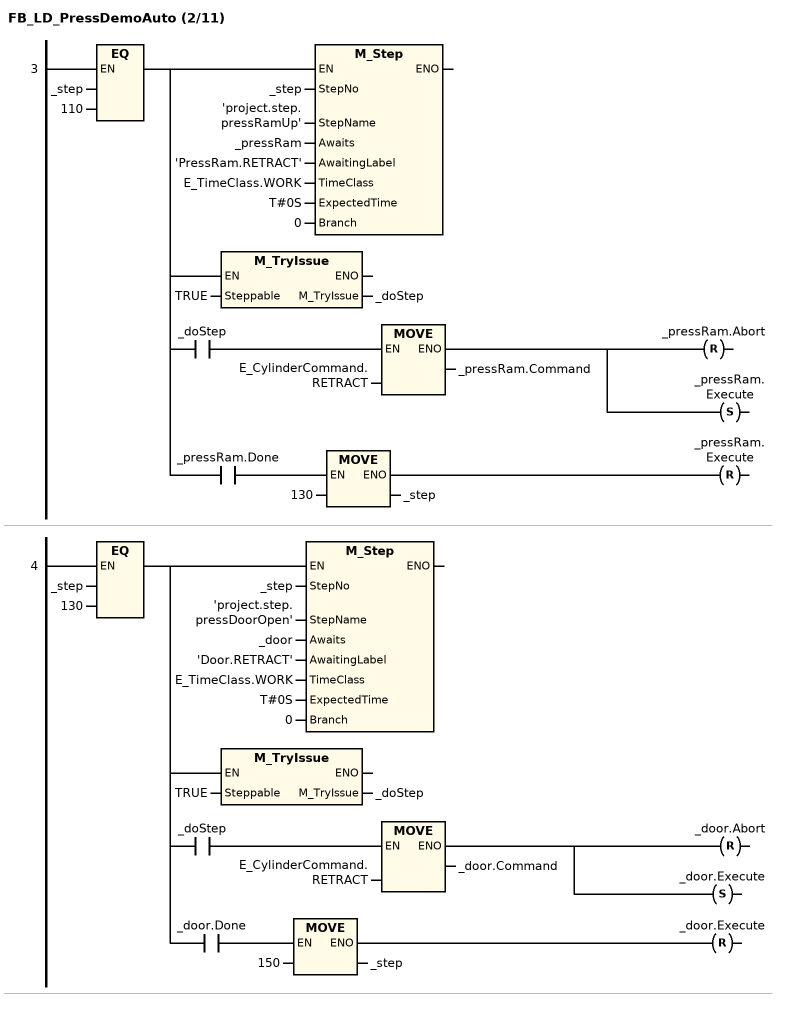
// NETWORK 3
_w5 := _step = 110;
IF _w5 THEN
    M_Step(StepNo := _step, StepName := 'project.step.pressRamUp', Awaits := _pressRam, AwaitingLabel := 'PressRam.RETRACT', TimeClass := E_TimeClass.WORK, ExpectedTime := T#0S, Branch := 0);
END_IF
IF _w5 THEN _doStep := M_TryIssue(Steppable := TRUE); END_IF
IF _w5 AND _doStep THEN _pressRam.Command := E_CylinderCommand.RETRACT; END_IF
_w6 := _w5 AND _doStep;
_pressRam.Abort R= _w6;
_pressRam.Execute S= _w6;
IF _w5 AND _pressRam.Done THEN _step := 130; END_IF
_pressRam.Execute R= _w5 AND _pressRam.Done;

// NETWORK 4
_w7 := _step = 130;
IF _w7 THEN
    M_Step(StepNo := _step, StepName := 'project.step.pressDoorOpen', Awaits := _door, AwaitingLabel := 'Door.RETRACT', TimeClass := E_TimeClass.WORK, ExpectedTime := T#0S, Branch := 0);
END_IF
IF _w7 THEN _doStep := M_TryIssue(Steppable := TRUE); END_IF
IF _w7 AND _doStep THEN _door.Command := E_CylinderCommand.RETRACT; END_IF
_w8 := _w7 AND _doStep;
_door.Abort R= _w8;
_door.Execute S= _w8;
IF _w7 AND _door.Done THEN _step := 150; END_IF
_door.Execute R= _w7 AND _door.Done;

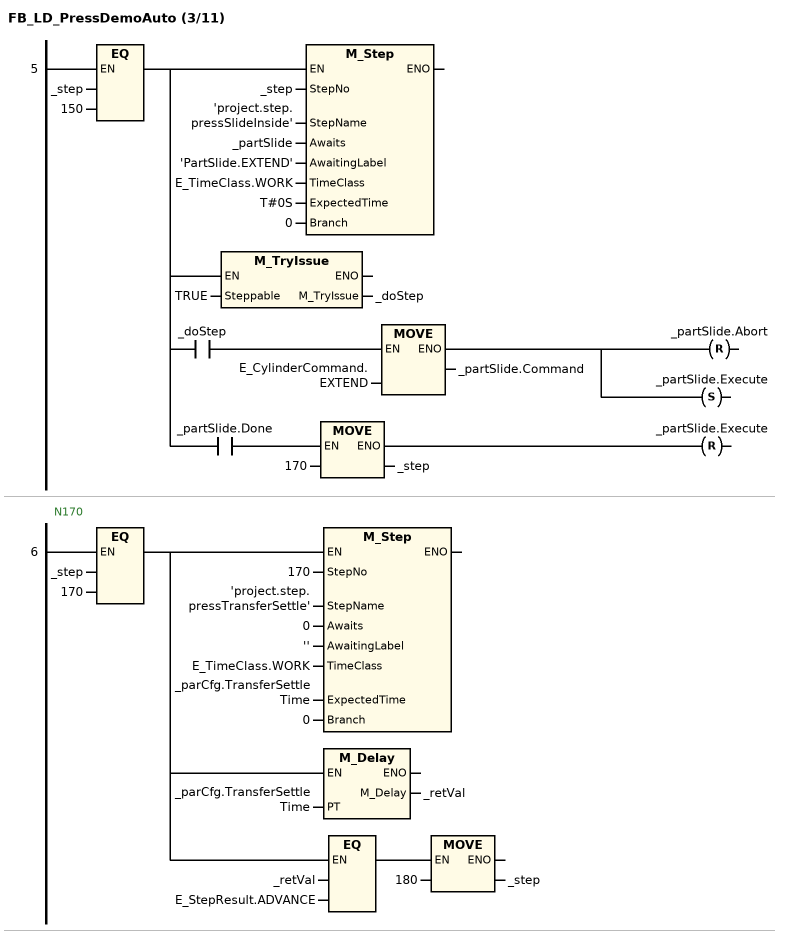
// NETWORK 5
_w9 := _step = 150;
IF _w9 THEN
    M_Step(StepNo := _step, StepName := 'project.step.pressSlideInside', Awaits := _partSlide, AwaitingLabel := 'PartSlide.EXTEND', TimeClass := E_TimeClass.WORK, ExpectedTime := T#0S, Branch := 0);
END_IF
IF _w9 THEN _doStep := M_TryIssue(Steppable := TRUE); END_IF
IF _w9 AND _doStep THEN _partSlide.Command := E_CylinderCommand.EXTEND; END_IF
_w10 := _w9 AND _doStep;
_partSlide.Abort R= _w10;
_partSlide.Execute S= _w10;
IF _w9 AND _partSlide.Done THEN _step := 170; END_IF
_partSlide.Execute R= _w9 AND _partSlide.Done;

// NETWORK 6
// N170
_w11 := _step = 170;
IF _w11 THEN
    M_Step(StepNo := 170, StepName := 'project.step.pressTransferSettle', Awaits := 0, AwaitingLabel := '', TimeClass := E_TimeClass.WORK, ExpectedTime := _parCfg.TransferSettleTime, Branch := 0);
END_IF
IF _w11 THEN _retVal := M_Delay(PT := _parCfg.TransferSettleTime); END_IF
IF _w11 AND _retVal = E_StepResult.ADVANCE THEN _step := 180; END_IF

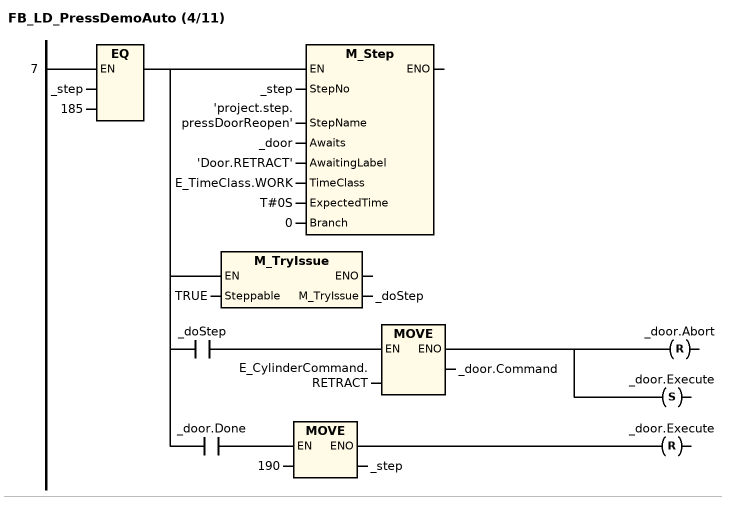
// NETWORK 7
_w12 := _step = 185;
IF _w12 THEN
    M_Step(StepNo := _step, StepName := 'project.step.pressDoorReopen', Awaits := _door, AwaitingLabel := 'Door.RETRACT', TimeClass := E_TimeClass.WORK, ExpectedTime := T#0S, Branch := 0);
END_IF
IF _w12 THEN _doStep := M_TryIssue(Steppable := TRUE); END_IF
IF _w12 AND _doStep THEN _door.Command := E_CylinderCommand.RETRACT; END_IF
_w13 := _w12 AND _doStep;
_door.Abort R= _w13;
_door.Execute S= _w13;
IF _w12 AND _door.Done THEN _step := 190; END_IF
_door.Execute R= _w12 AND _door.Done;

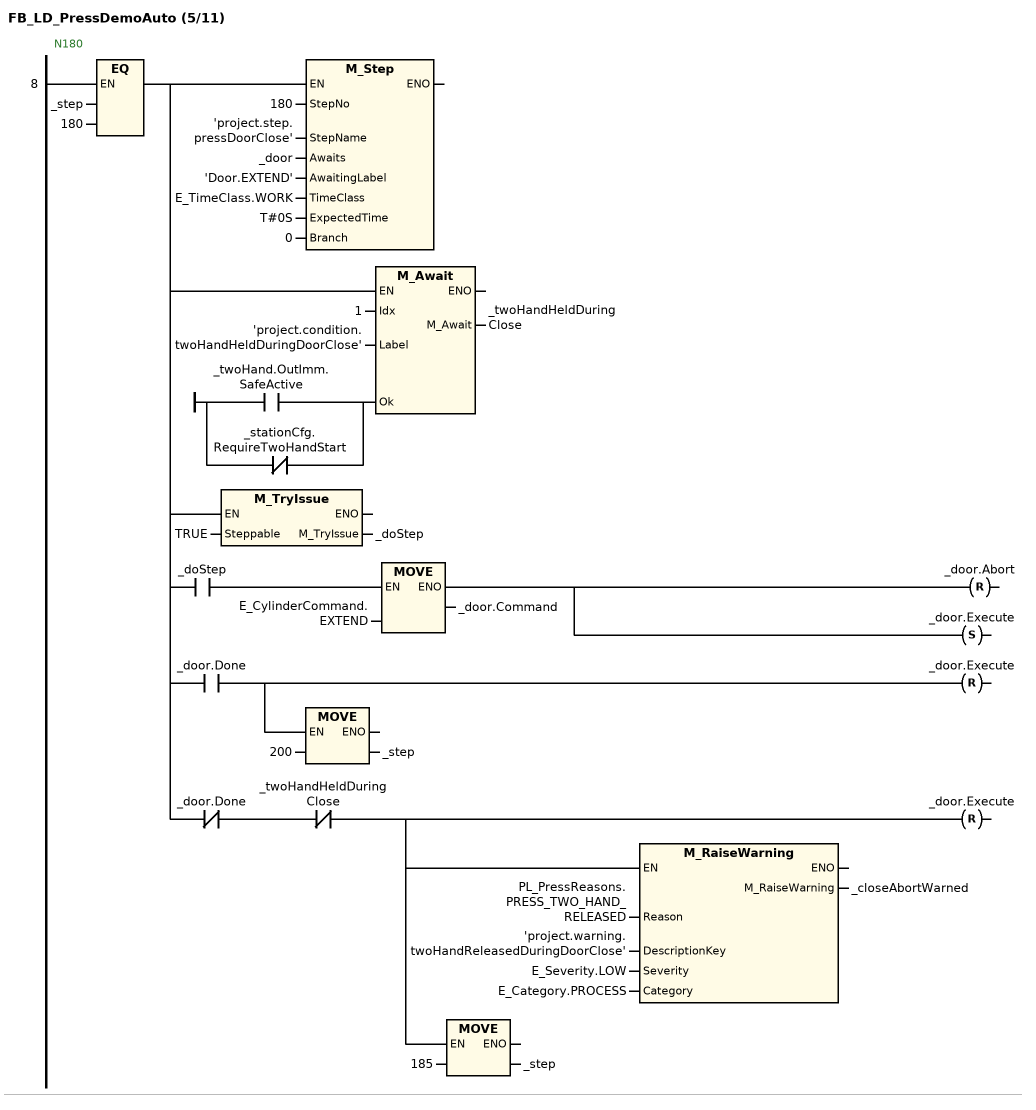
// NETWORK 8
// N180
_w14 := _step = 180;
IF _w14 THEN
    M_Step(StepNo := 180, StepName := 'project.step.pressDoorClose', Awaits := _door, AwaitingLabel := 'Door.EXTEND', TimeClass := E_TimeClass.WORK, ExpectedTime := T#0S, Branch := 0);
END_IF
IF _w14 THEN
    _twoHandHeldDuringClose := M_Await(Idx := 1, Label := 'project.condition.twoHandHeldDuringDoorClose', Ok := _twoHand.OutImm.SafeActive OR NOT _stationCfg.RequireTwoHandStart);
END_IF
IF _w14 THEN _doStep := M_TryIssue(Steppable := TRUE); END_IF
IF _w14 AND _doStep THEN _door.Command := E_CylinderCommand.EXTEND; END_IF
_w15 := _w14 AND _doStep;
_door.Abort R= _w15;
_door.Execute S= _w15;
_w16 := _w14 AND _door.Done;
_door.Execute R= _w16;
IF _w16 THEN _step := 200; END_IF
_w17 := _w14 AND NOT _door.Done AND NOT _twoHandHeldDuringClose;
_door.Execute R= _w17;
IF _w17 THEN
    _closeAbortWarned := M_RaiseWarning(Reason := PL_PressReasons.PRESS_TWO_HAND_RELEASED, DescriptionKey := 'project.warning.twoHandReleasedDuringDoorClose', Severity := E_Severity.LOW, Category := E_Category.PROCESS);
END_IF
IF _w17 THEN _step := 185; END_IF

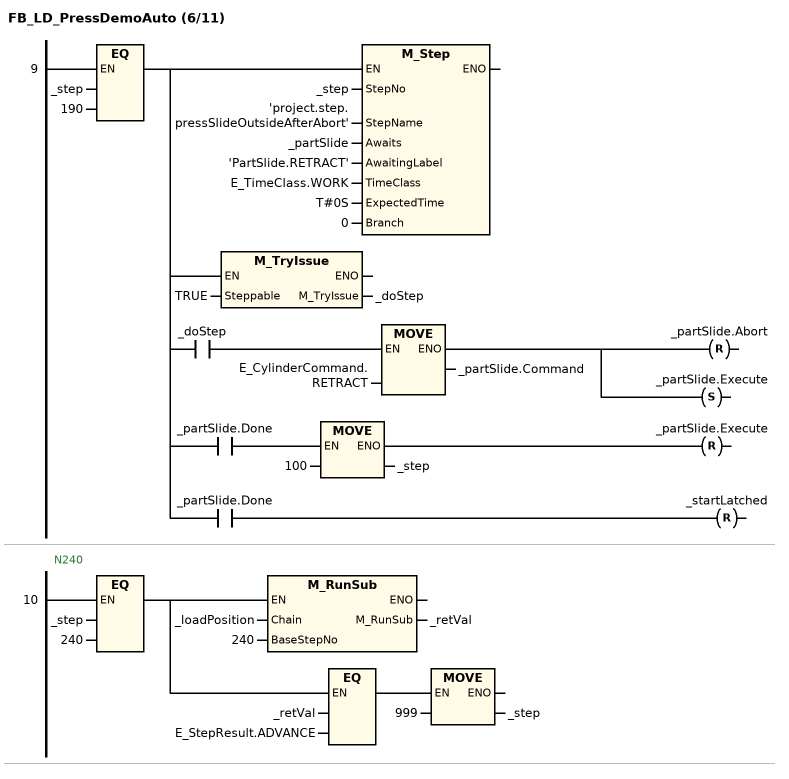
// NETWORK 9
_w18 := _step = 190;
IF _w18 THEN
    M_Step(StepNo := _step, StepName := 'project.step.pressSlideOutsideAfterAbort', Awaits := _partSlide, AwaitingLabel := 'PartSlide.RETRACT', TimeClass := E_TimeClass.WORK, ExpectedTime := T#0S, Branch := 0);
END_IF
IF _w18 THEN _doStep := M_TryIssue(Steppable := TRUE); END_IF
IF _w18 AND _doStep THEN _partSlide.Command := E_CylinderCommand.RETRACT; END_IF
_w19 := _w18 AND _doStep;
_partSlide.Abort R= _w19;
_partSlide.Execute S= _w19;
IF _w18 AND _partSlide.Done THEN _step := 100; END_IF
_partSlide.Execute R= _w18 AND _partSlide.Done;
_startLatched R= _w18 AND _partSlide.Done;

// NETWORK 10
// N240
_w20 := _step = 240;
IF _w20 THEN _retVal := M_RunSub(Chain := _loadPosition, BaseStepNo := 240); END_IF
IF _w20 AND _retVal = E_StepResult.ADVANCE THEN _step := 999; END_IF

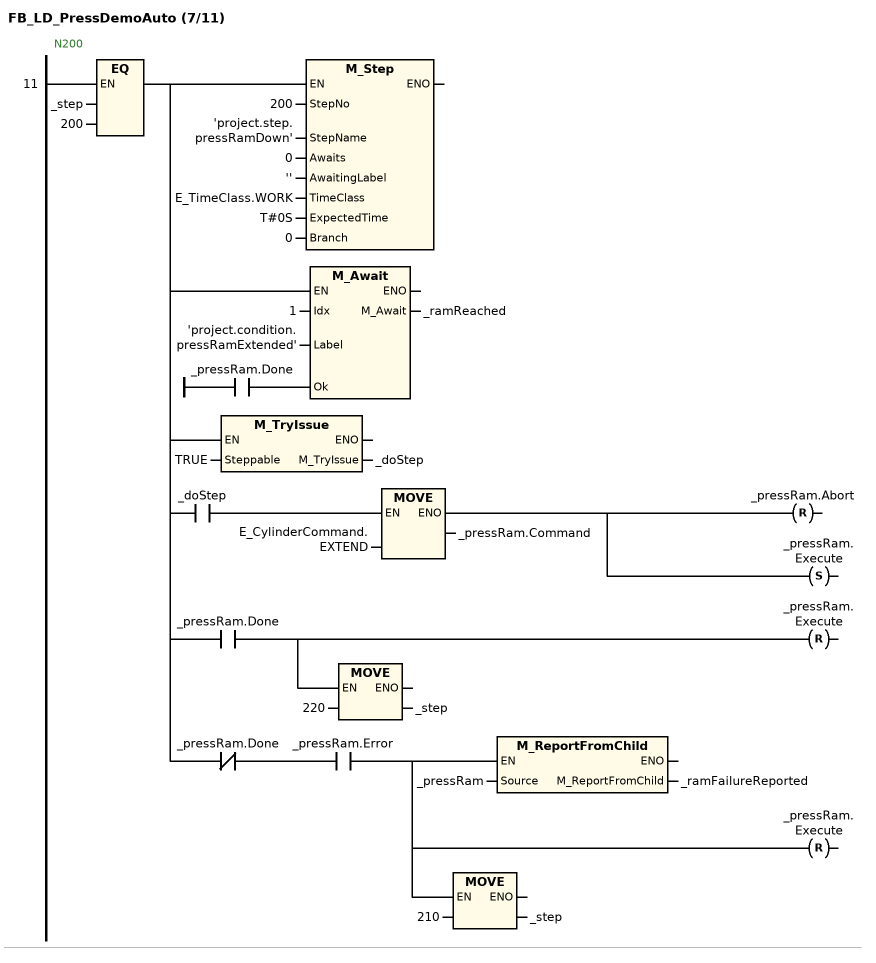
// NETWORK 11
// N200
_w21 := _step = 200;
IF _w21 THEN
    M_Step(StepNo := 200, StepName := 'project.step.pressRamDown', Awaits := 0, AwaitingLabel := '', TimeClass := E_TimeClass.WORK, ExpectedTime := T#0S, Branch := 0);
END_IF
IF _w21 THEN
    _ramReached := M_Await(Idx := 1, Label := 'project.condition.pressRamExtended', Ok := _pressRam.Done);
END_IF
IF _w21 THEN _doStep := M_TryIssue(Steppable := TRUE); END_IF
IF _w21 AND _doStep THEN _pressRam.Command := E_CylinderCommand.EXTEND; END_IF
_w22 := _w21 AND _doStep;
_pressRam.Abort R= _w22;
_pressRam.Execute S= _w22;
_w23 := _w21 AND _pressRam.Done;
_pressRam.Execute R= _w23;
IF _w23 THEN _step := 220; END_IF
_w24 := _w21 AND NOT _pressRam.Done AND _pressRam.Error;
IF _w24 THEN _ramFailureReported := M_ReportFromChild(Source := _pressRam); END_IF
_pressRam.Execute R= _w24;
IF _w24 THEN _step := 210; END_IF

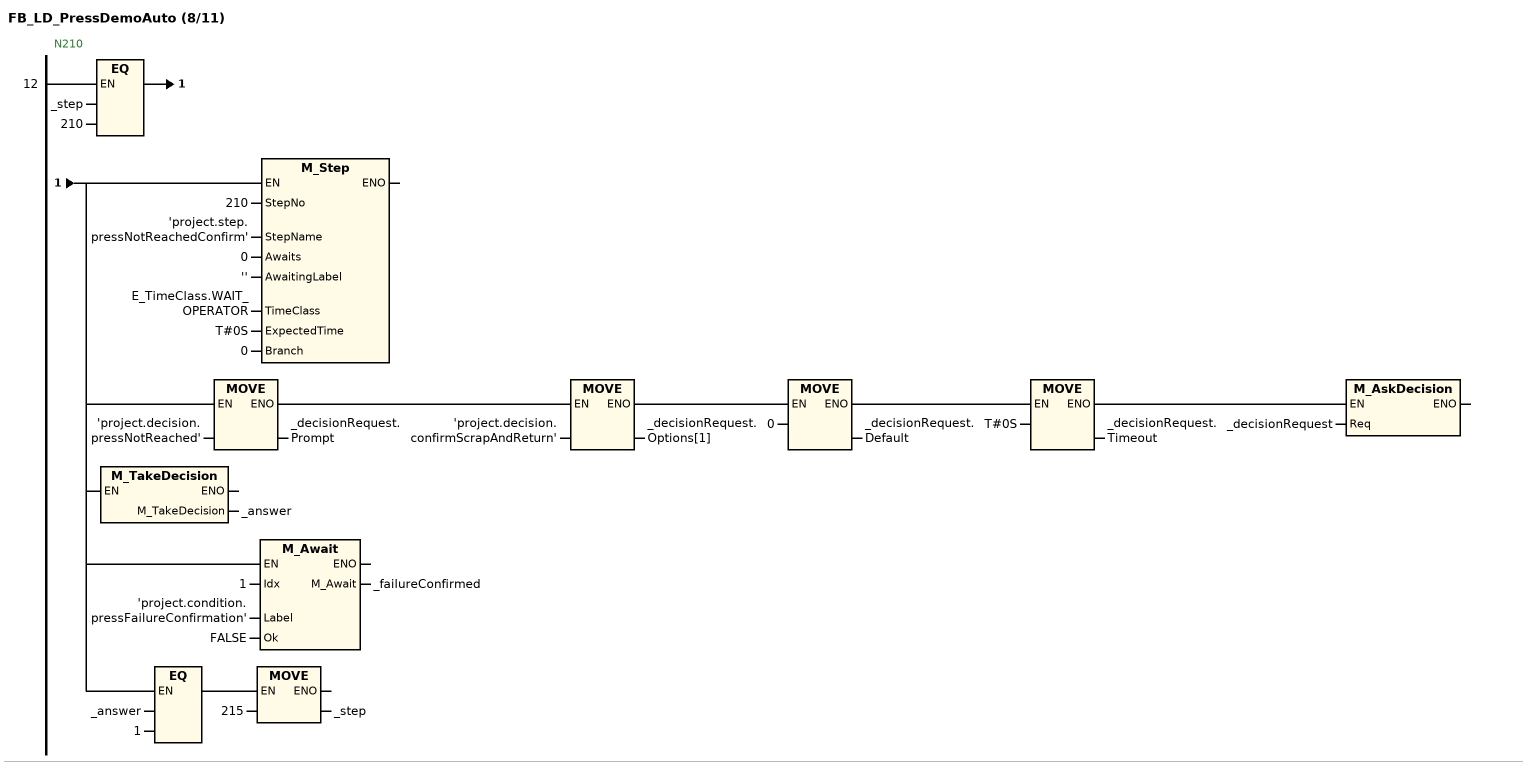
// NETWORK 12
// N210
_w25 := _step = 210;
IF _w25 THEN
    M_Step(StepNo := 210, StepName := 'project.step.pressNotReachedConfirm', Awaits := 0, AwaitingLabel := '', TimeClass := E_TimeClass.WAIT_OPERATOR, ExpectedTime := T#0S, Branch := 0);
END_IF
IF _w25 THEN _decisionRequest.Prompt := 'project.decision.pressNotReached'; END_IF
IF _w25 THEN _decisionRequest.Options[1] := 'project.decision.confirmScrapAndReturn'; END_IF
IF _w25 THEN _decisionRequest.Default := 0; END_IF
IF _w25 THEN _decisionRequest.Timeout := T#0S; END_IF
IF _w25 THEN M_AskDecision(Req := _decisionRequest); END_IF
IF _w25 THEN _answer := M_TakeDecision(); END_IF
IF _w25 THEN
    _failureConfirmed := M_Await(Idx := 1, Label := 'project.condition.pressFailureConfirmation', Ok := FALSE);
END_IF
IF _w25 AND _answer = 1 THEN _step := 215; END_IF

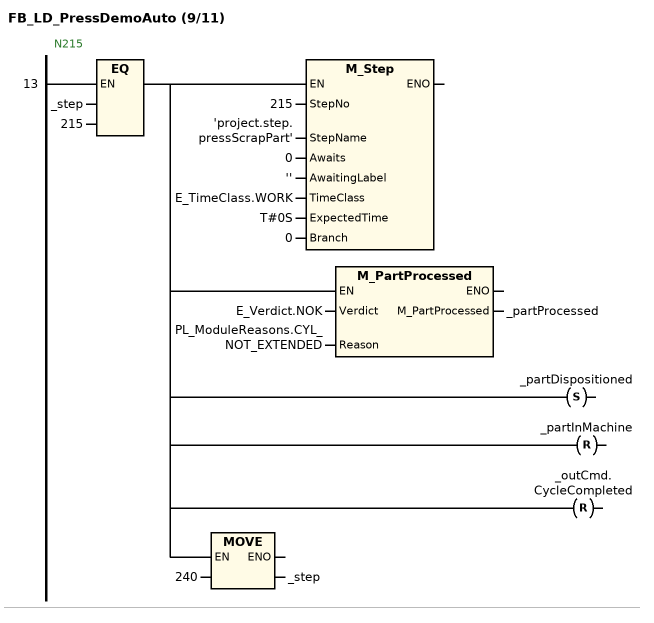
// NETWORK 13
// N215
_w26 := _step = 215;
IF _w26 THEN
    M_Step(StepNo := 215, StepName := 'project.step.pressScrapPart', Awaits := 0, AwaitingLabel := '', TimeClass := E_TimeClass.WORK, ExpectedTime := T#0S, Branch := 0);
END_IF
IF _w26 THEN
    _partProcessed := M_PartProcessed(Verdict := E_Verdict.NOK, Reason := PL_ModuleReasons.CYL_NOT_EXTENDED);
END_IF
_partDispositioned S= _w26;
_partInMachine R= _w26;
_outCmd.CycleCompleted R= _w26;
IF _w26 THEN _step := 240; END_IF

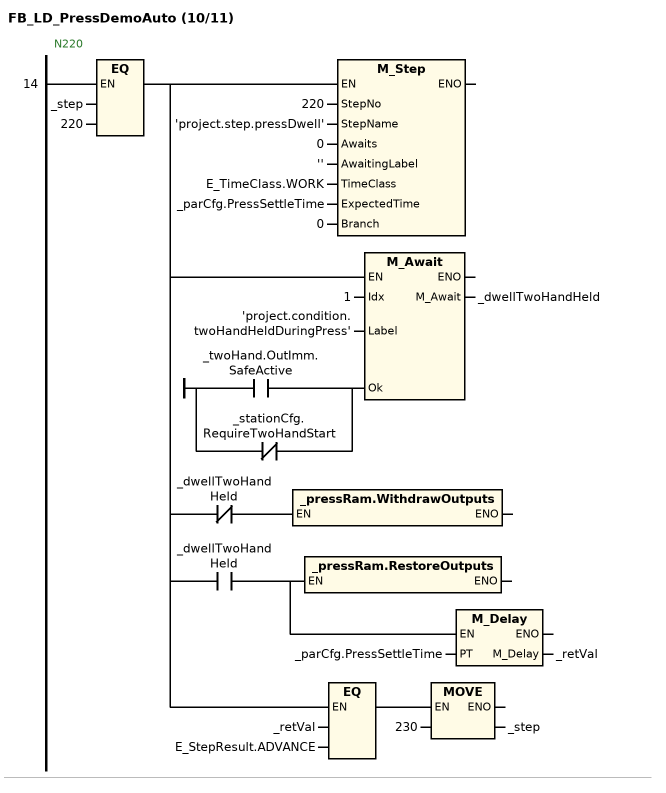
// NETWORK 14
// N220
_w27 := _step = 220;
IF _w27 THEN
    M_Step(StepNo := 220, StepName := 'project.step.pressDwell', Awaits := 0, AwaitingLabel := '', TimeClass := E_TimeClass.WORK, ExpectedTime := _parCfg.PressSettleTime, Branch := 0);
END_IF
IF _w27 THEN
    _dwellTwoHandHeld := M_Await(Idx := 1, Label := 'project.condition.twoHandHeldDuringPress', Ok := _twoHand.OutImm.SafeActive OR NOT _stationCfg.RequireTwoHandStart);
END_IF
IF _w27 AND NOT _dwellTwoHandHeld THEN _pressRam.WithdrawOutputs(); END_IF
_w28 := _w27 AND _dwellTwoHandHeld;
IF _w28 THEN _pressRam.RestoreOutputs(); END_IF
IF _w28 THEN _retVal := M_Delay(PT := _parCfg.PressSettleTime); END_IF
IF _w27 AND _retVal = E_StepResult.ADVANCE THEN _step := 230; END_IF

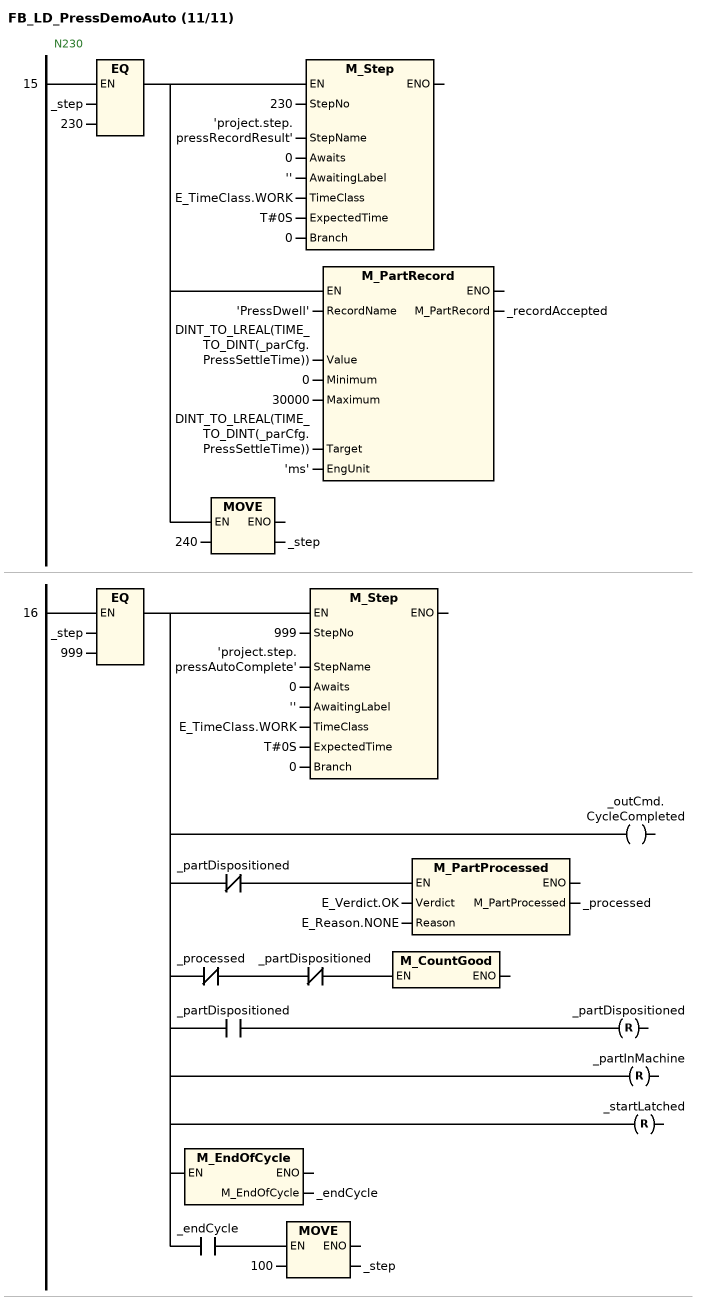
// NETWORK 15
// N230
_w29 := _step = 230;
IF _w29 THEN
    M_Step(StepNo := 230, StepName := 'project.step.pressRecordResult', Awaits := 0, AwaitingLabel := '', TimeClass := E_TimeClass.WORK, ExpectedTime := T#0S, Branch := 0);
END_IF
IF _w29 THEN
    _recordAccepted := M_PartRecord(RecordName := 'PressDwell', Value := DINT_TO_LREAL(TIME_TO_DINT(_parCfg.PressSettleTime)), Minimum := 0, Maximum := 30000, Target := DINT_TO_LREAL(TIME_TO_DINT(_parCfg.PressSettleTime)), EngUnit := 'ms');
END_IF
IF _w29 THEN _step := 240; END_IF

// NETWORK 16
_w30 := _step = 999;
IF _w30 THEN
    M_Step(StepNo := 999, StepName := 'project.step.pressAutoComplete', Awaits := 0, AwaitingLabel := '', TimeClass := E_TimeClass.WORK, ExpectedTime := T#0S, Branch := 0);
END_IF
_outCmd.CycleCompleted := _w30;
IF _w30 AND NOT _partDispositioned THEN
    _processed := M_PartProcessed(Verdict := E_Verdict.OK, Reason := E_Reason.NONE);
END_IF
IF _w30 AND NOT _processed AND NOT _partDispositioned THEN M_CountGood(); END_IF
_partDispositioned R= _w30 AND _partDispositioned;
_partInMachine R= _w30;
_startLatched R= _w30;
IF _w30 THEN _endCycle := M_EndOfCycle(); END_IF
IF _w30 AND _endCycle THEN _step := 100; END_IF

// Identical signature to the ST and SFC renditions of this chain, so the Unit can
// bind whichever one AUTO_SEQUENCE_LANGUAGE selects without any other difference.
METHOD Setup : BOOL
VAR_INPUT
    Host : I_SequenceHost;
END_VAR
VAR_IN_OUT
    PressRam : FB_CylinderCM;
    Door : FB_CylinderCM;
    PartSlide : FB_CylinderCM;
    TwoHand : FB_TwoHandStartCM;
    PartPresentSensor : FB_DigitalInputCM;
    AirPressureMonitor : FB_AirPressureMonitorCM;
    ParCfg : ST_PneumaticPressParCfg;
    StationCfg : ST_PneumaticPressStationCfg;
    OutCmd : ST_PneumaticPressOutCmd;
    StartLatched : BOOL;
END_VAR
_pressRam REF= PressRam;
_door REF= Door;
_partSlide REF= PartSlide;
_twoHand REF= TwoHand;
_partPresentSensor REF= PartPresentSensor;
_airPressureMonitor REF= AirPressureMonitor;
_parCfg REF= ParCfg;
_stationCfg REF= StationCfg;
_outCmd REF= OutCmd;
_startLatched REF= StartLatched;
Setup := M_Attach(Host := Host) AND __ISVALIDREF(_pressRam) AND __ISVALIDREF(_door)
    AND __ISVALIDREF(_partSlide) AND __ISVALIDREF(_twoHand)
    AND __ISVALIDREF(_partPresentSensor) AND __ISVALIDREF(_airPressureMonitor)
    AND __ISVALIDREF(_parCfg) AND __ISVALIDREF(_outCmd) AND __ISVALIDREF(_startLatched)
    AND _loadPosition.Setup(Host := Host, PressRam := PressRam, Door := Door, PartSlide := PartSlide);
END_METHOD

// §6.8 - the chain's own state on a restart (the base resets the flow state).
METHOD PROTECTED OnChainReset
// A chart restart abandons whatever the cycle was holding: the part record is
// closed by N215/N999, never by a restart, so both trackers start clean.
_partDispositioned := FALSE;
_partInMachine := FALSE;
END_METHOD

END_FUNCTION_BLOCK

// ---- Fraktal_Press_Demo/01_PneumaticPress/Release/FB_PressDemoRelease.TcPOU
// Project-owned release engineering for the pneumatic press.
// This FB is not a Fraktal module: it exposes named condition state and fills
// the Unit's authoritative release reports without adding an OPC UA tree node.
FUNCTION_BLOCK FB_PressDemoRelease EXTENDS FB_PressDemoReleaseState
VAR
    _ramExtendOk : BOOL;
    _ramExtendKey : STRING(255);
END_VAR

; // Evaluated explicitly by the owning Unit after child cyclic status is available.

METHOD Setup : BOOL
VAR_INPUT
    UnitPath : STRING(255);
END_VAR
_unitPath := UnitPath;
Setup := ModeStart.Define(Index := 1, Description := 'project.condition.airPressureOk',
    Reason := E_Reason.PERMISSIVE_NOT_MET, Bypassable := FALSE);
END_METHOD

METHOD M_Evaluate
VAR_INPUT
    PressRam : REFERENCE TO FB_CylinderCM;
    Door : REFERENCE TO FB_CylinderCM;
    PartSlide : REFERENCE TO FB_CylinderCM;
    TwoHand : REFERENCE TO FB_TwoHandStartCM;
    PneumaticPower : REFERENCE TO FB_PowerGroupCM;
    AirPressure : REFERENCE TO FB_AirPressureMonitorCM;
END_VAR
// Direction-specific functional collision prevention. Certified safety remains
// authoritative for hazardous-motion permission and safe output removal.
Door.SetDirectionalPermits(
    ExtendOk := PartSlide.OutImm.Extended AND NOT PartSlide.OutImm.Retracted
        AND NOT PartSlide.Busy AND NOT PartSlide.Error,
    RetractOk := TRUE,
    ExtendDescriptionKey := 'project.interlock.doorCloseRequiresSlideInside',
    RetractDescriptionKey := 'project.interlock.doorOpenPermitted');
PartSlide.SetDirectionalPermits(
    ExtendOk := Door.OutImm.Retracted AND NOT Door.OutImm.Extended
        AND NOT Door.Busy AND NOT Door.Error,
    RetractOk := Door.OutImm.Retracted AND NOT Door.OutImm.Extended
        AND NOT Door.Busy AND NOT Door.Error,
    ExtendDescriptionKey := 'project.interlock.slideMoveRequiresDoorOpen',
    RetractDescriptionKey := 'project.interlock.slideOutsideRequiresDoorOpen');
// Evaluate each ram-extend condition by name, then report the FIRST one that is
// missing (Core Sec.6.9 first-out). SetDirectionalPermits carries one key per
// direction, so the first-out choice is made here rather than losing it.
RamGuardClosed    := Door.OutImm.Extended AND NOT Door.OutImm.Retracted;
RamSlideInside    := PartSlide.OutImm.Extended AND NOT PartSlide.OutImm.Retracted;
RamDevicesHealthy := NOT Door.Error AND NOT PartSlide.Error;
RamAirPressureOk  := AirPressure.OutImm.PressureOk;
RamTwoHandHeld    := TwoHand.OutImm.SafeActive;
RamControlPowerOn := PneumaticPower.OutCmd.PowerOn;
_ramExtendOk := RamGuardClosed AND RamSlideInside AND RamDevicesHealthy
    AND RamAirPressureOk AND RamTwoHandHeld AND RamControlPowerOn;

IF NOT RamControlPowerOn THEN
    _ramExtendKey := 'project.interlock.pressRequiresControlPower';
ELSIF NOT RamAirPressureOk THEN
    _ramExtendKey := 'project.interlock.pressRequiresAirPressure';
ELSIF NOT RamGuardClosed THEN
    _ramExtendKey := 'project.interlock.pressRequiresGuardClosed';
ELSIF NOT RamSlideInside THEN
    _ramExtendKey := 'project.interlock.pressRequiresSlideInside';
ELSIF NOT RamDevicesHealthy THEN
    _ramExtendKey := 'project.interlock.pressRequiresHealthyGuardSlide';
ELSIF NOT RamTwoHandHeld THEN
    _ramExtendKey := 'project.interlock.pressRequiresTwoHandHeld';
ELSE
    _ramExtendKey := 'project.interlock.pressRamExtendPermitted';
END_IF

PressRam.SetDirectionalPermits(
    ExtendOk := _ramExtendOk,
    RetractOk := TRUE,
    ExtendDescriptionKey := _ramExtendKey,
    RetractDescriptionKey := 'project.interlock.pressRetractPermitted');

// Mode-entry release is distinct from future AUTO waits. Part presence and the
// two-hand edge remain live conditions in the AUTO SFC action.
ModeStartAirPressureOk := AirPressure.OutImm.PressureOk;
ModeStart.Cond[1] := ModeStartAirPressureOk;
ModeStart();
END_METHOD

METHOD M_AppendStart
VAR_IN_OUT
    Report : ST_ReleaseReport;
END_VAR
ModeStart.AppendFailed(SourcePath := _unitPath, Report := Report);
END_METHOD

METHOD M_AppendManual
VAR_INPUT
    TargetPath : STRING(255);
    Value : DINT;
    PressRam : REFERENCE TO FB_CylinderCM;
    Door : REFERENCE TO FB_CylinderCM;
    PartSlide : REFERENCE TO FB_CylinderCM;
END_VAR
VAR_IN_OUT
    Report : ST_ReleaseReport;
END_VAR
IF TargetPath = PressRam.Name THEN
    PressRam.AppendDirectionalRelease(Value := Value, Report := Report);
ELSIF TargetPath = Door.Name THEN
    Door.AppendDirectionalRelease(Value := Value, Report := Report);
ELSIF TargetPath = PartSlide.Name THEN
    PartSlide.AppendDirectionalRelease(Value := Value, Report := Report);
ELSE
    IF Report.Count < PL_Fraktal.MAX_RELEASE_REASONS THEN
        Report.Count := Report.Count + 1;
        Report.Reasons[Report.Count].Description := 'std.error.unsupportedManualTarget';
        Report.Reasons[Report.Count].ReasonCode := E_Reason.UNSUPPORTED_COMMAND;
        Report.Reasons[Report.Count].SourcePath := _unitPath;
        Report.Reasons[Report.Count].Kind := E_ReleaseKind.OTHER;
        Report.Reasons[Report.Count].Bypassable := FALSE;
    ELSE
        ; // bounded report is full; no array write is attempted
    END_IF
END_IF
END_METHOD

END_FUNCTION_BLOCK

// ---- Fraktal_Press_Demo/01_PneumaticPress/Release/FB_PressDemoReleaseState.TcPOU
// The state the press's two release renditions (ST FB_PressDemoRelease, LD
// FB_LD_PressDemoRelease) share. Both declared this block word for word; it is
// declared once here and each rendition keeps only its LOGIC, which is the
// part the bench exists to carry twice (§1.1 O9). Not a Fraktal module.
FUNCTION_BLOCK FB_PressDemoReleaseState
VAR_OUTPUT
    ModeStart : FB_PermIntlk;
    ModeStartAirPressureOk : BOOL;
    // Ram-extend permissive, split into individually named conditions. A single
    // composite permit could only ever report one composite key, so releasing
    // the two-hand button - the NORMAL way an operator stops a stroke - was
    // indistinguishable from a guard fault, an air loss or a power loss.
    RamGuardClosed   : BOOL;
    RamSlideInside   : BOOL;
    RamDevicesHealthy: BOOL;
    RamAirPressureOk : BOOL;
    RamTwoHandHeld   : BOOL;
    RamControlPowerOn: BOOL;
END_VAR
VAR
    _unitPath : STRING(255);
END_VAR

;

// Copy the evaluated conditions into the Unit's published record. Called for
// the SELECTED rendition only, straight after it evaluated, every scan.
METHOD M_PublishTo
VAR_IN_OUT
    Conditions : ST_PressDemoReleaseConditions;
END_VAR
Conditions.ModeStartAirPressureOk := ModeStartAirPressureOk;
Conditions.RamGuardClosed := RamGuardClosed;
Conditions.RamSlideInside := RamSlideInside;
Conditions.RamDevicesHealthy := RamDevicesHealthy;
Conditions.RamAirPressureOk := RamAirPressureOk;
Conditions.RamTwoHandHeld := RamTwoHandHeld;
Conditions.RamControlPowerOn := RamControlPowerOn;
END_METHOD

END_FUNCTION_BLOCK

// ---- Fraktal_Press_Demo/01_PneumaticPress/Release/FB_LD_PressDemoRelease.TcPOU
// Project-owned release engineering for the pneumatic press, authored in LADDER.
//
// This is an O2 DEMONSTRATION IN THE BENCH, not a per-project pattern. Core
// §6.8/§7.2 permit a sequence or an interlock to be authored in ST, SFC or LD,
// and the only way that claim is testable is to carry a rendition and compile
// it. Two renditions of one interlock is duplication §1.1 O9 would otherwise
// forbid outright - it is justified here, and ONLY here, because demonstrating
// the language choice IS this project's purpose, exactly as the three AUTO
// chain renditions are. A real project writes this once, in one language.
// FB_PressDemoUnit.RELEASE_LANGUAGE selects which one is evaluated.
//
// Same public surface as FB_PressDemoRelease so the Unit binds either without
// any other difference, and like it this is not a Fraktal module: it exposes
// named condition state and fills the Unit's authoritative release reports
// without adding an OPC UA tree node.
FUNCTION_BLOCK FB_LD_PressDemoRelease EXTENDS FB_PressDemoReleaseState
VAR
    _ramExtendOk : BOOL;
    _ramExtendKey : STRING(255);
    // AppendFailed returns the new report count. ST may discard a return value;
    // a rung has to land it somewhere, and the ENO slot is not that somewhere.
    _appendCount : INT;
END_VAR

; // Evaluated explicitly by the owning Unit after child cyclic status is available.

METHOD Setup : BOOL
VAR_INPUT
    UnitPath : STRING(255);
END_VAR
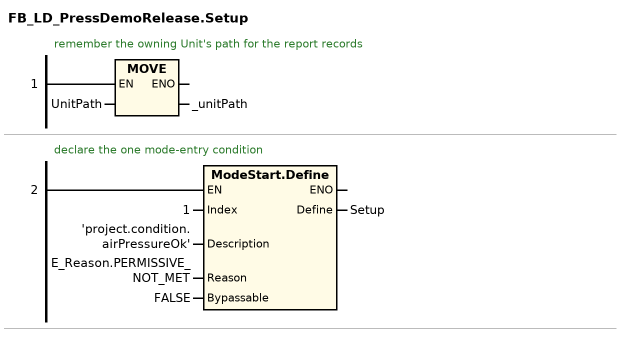
// NETWORK 1
// remember the owning Unit's path for the report records
_unitPath := UnitPath;

// NETWORK 2
// declare the one mode-entry condition
Setup := ModeStart.Define(Index := 1, Description := 'project.condition.airPressureOk', Reason := E_Reason.PERMISSIVE_NOT_MET, Bypassable := FALSE);
END_METHOD

METHOD M_Evaluate
VAR_INPUT
    PressRam : REFERENCE TO FB_CylinderCM;
    Door : REFERENCE TO FB_CylinderCM;
    PartSlide : REFERENCE TO FB_CylinderCM;
    TwoHand : REFERENCE TO FB_TwoHandStartCM;
    PneumaticPower : REFERENCE TO FB_PowerGroupCM;
    AirPressure : REFERENCE TO FB_AirPressureMonitorCM;
END_VAR
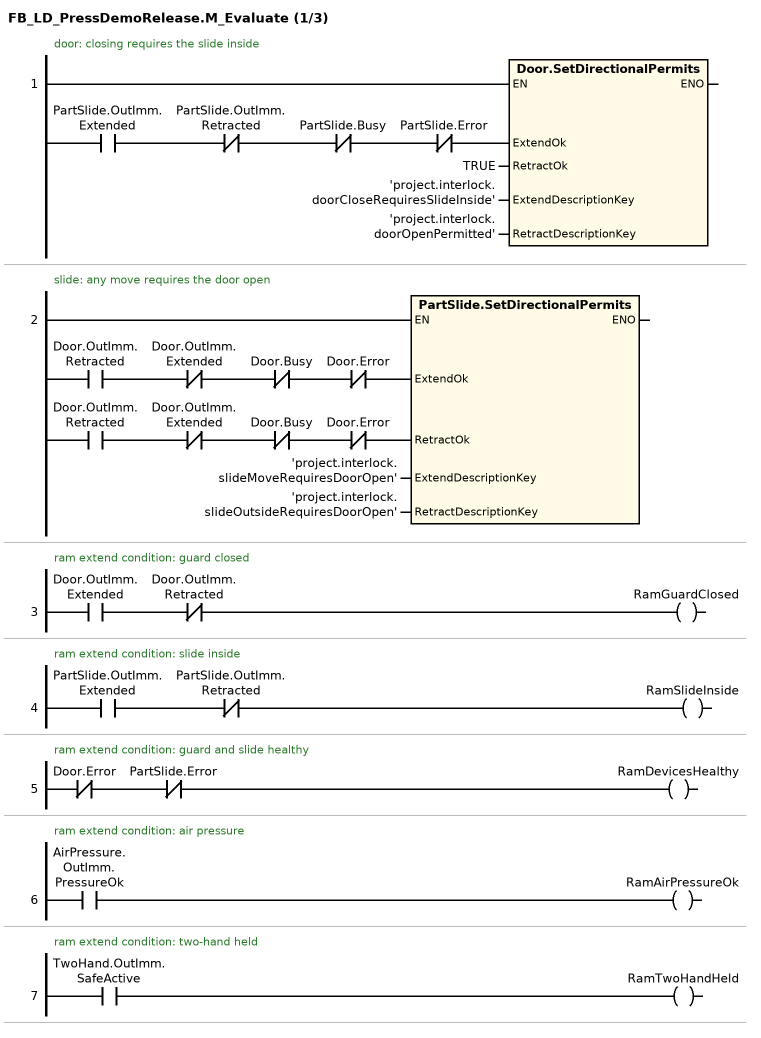
// NETWORK 1
// door: closing requires the slide inside
Door.SetDirectionalPermits(ExtendOk := PartSlide.OutImm.Extended AND NOT PartSlide.OutImm.Retracted AND NOT PartSlide.Busy AND NOT PartSlide.Error, RetractOk := TRUE, ExtendDescriptionKey := 'project.interlock.doorCloseRequiresSlideInside', RetractDescriptionKey := 'project.interlock.doorOpenPermitted');

// NETWORK 2
// slide: any move requires the door open
PartSlide.SetDirectionalPermits(ExtendOk := Door.OutImm.Retracted AND NOT Door.OutImm.Extended AND NOT Door.Busy AND NOT Door.Error, RetractOk := Door.OutImm.Retracted AND NOT Door.OutImm.Extended AND NOT Door.Busy AND NOT Door.Error, ExtendDescriptionKey := 'project.interlock.slideMoveRequiresDoorOpen', RetractDescriptionKey := 'project.interlock.slideOutsideRequiresDoorOpen');

// NETWORK 3
// ram extend condition: guard closed
RamGuardClosed := Door.OutImm.Extended AND NOT Door.OutImm.Retracted;

// NETWORK 4
// ram extend condition: slide inside
RamSlideInside := PartSlide.OutImm.Extended AND NOT PartSlide.OutImm.Retracted;

// NETWORK 5
// ram extend condition: guard and slide healthy
RamDevicesHealthy := NOT Door.Error AND NOT PartSlide.Error;

// NETWORK 6
// ram extend condition: air pressure
RamAirPressureOk := AirPressure.OutImm.PressureOk;

// NETWORK 7
// ram extend condition: two-hand held
RamTwoHandHeld := TwoHand.OutImm.SafeActive;

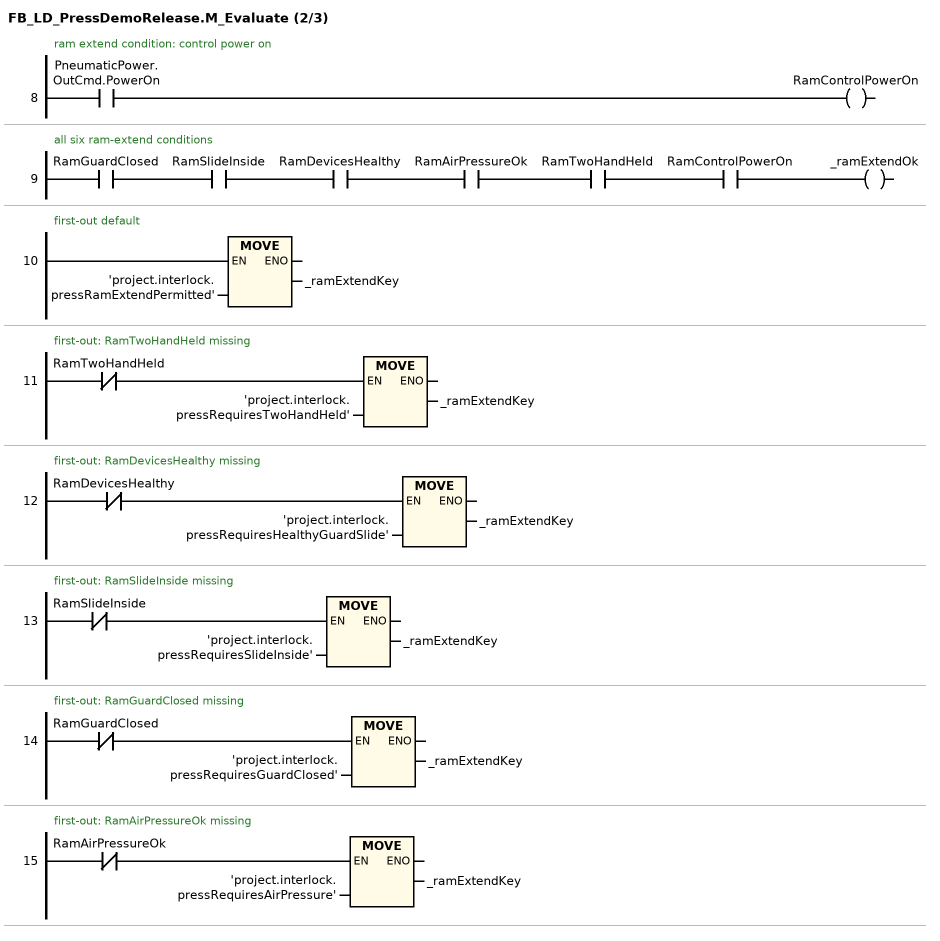
// NETWORK 8
// ram extend condition: control power on
RamControlPowerOn := PneumaticPower.OutCmd.PowerOn;

// NETWORK 9
// all six ram-extend conditions
_ramExtendOk := RamGuardClosed AND RamSlideInside AND RamDevicesHealthy AND RamAirPressureOk AND RamTwoHandHeld AND RamControlPowerOn;

// NETWORK 10
// first-out default
_ramExtendKey := 'project.interlock.pressRamExtendPermitted';

// NETWORK 11
// first-out: RamTwoHandHeld missing
IF NOT RamTwoHandHeld THEN _ramExtendKey := 'project.interlock.pressRequiresTwoHandHeld'; END_IF

// NETWORK 12
// first-out: RamDevicesHealthy missing
IF NOT RamDevicesHealthy THEN _ramExtendKey := 'project.interlock.pressRequiresHealthyGuardSlide'; END_IF

// NETWORK 13
// first-out: RamSlideInside missing
IF NOT RamSlideInside THEN _ramExtendKey := 'project.interlock.pressRequiresSlideInside'; END_IF

// NETWORK 14
// first-out: RamGuardClosed missing
IF NOT RamGuardClosed THEN _ramExtendKey := 'project.interlock.pressRequiresGuardClosed'; END_IF

// NETWORK 15
// first-out: RamAirPressureOk missing
IF NOT RamAirPressureOk THEN _ramExtendKey := 'project.interlock.pressRequiresAirPressure'; END_IF

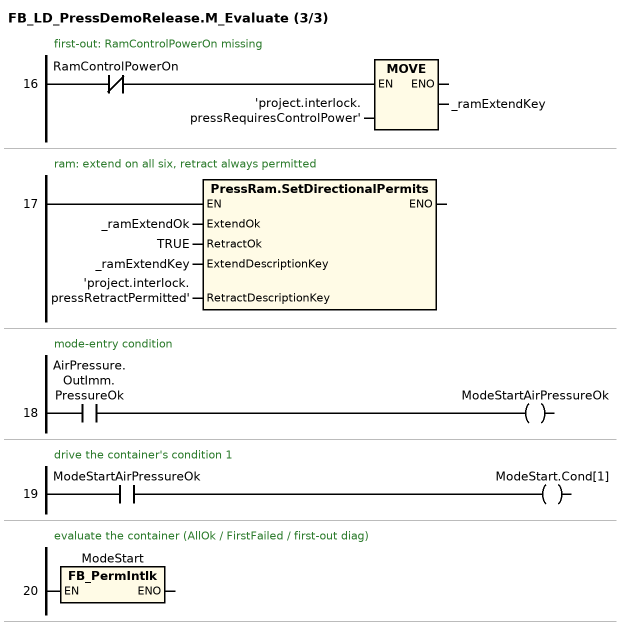
// NETWORK 16
// first-out: RamControlPowerOn missing
IF NOT RamControlPowerOn THEN _ramExtendKey := 'project.interlock.pressRequiresControlPower'; END_IF

// NETWORK 17
// ram: extend on all six, retract always permitted
PressRam.SetDirectionalPermits(ExtendOk := _ramExtendOk, RetractOk := TRUE, ExtendDescriptionKey := _ramExtendKey, RetractDescriptionKey := 'project.interlock.pressRetractPermitted');

// NETWORK 18
// mode-entry condition
ModeStartAirPressureOk := AirPressure.OutImm.PressureOk;

// NETWORK 19
// drive the container's condition 1
ModeStart.Cond[1] := ModeStartAirPressureOk;

// NETWORK 20
// evaluate the container (AllOk / FirstFailed / first-out diag)
ModeStart(); // FB_PermIntlk
END_METHOD

METHOD M_AppendStart
VAR_IN_OUT
    Report : ST_ReleaseReport;
END_VAR
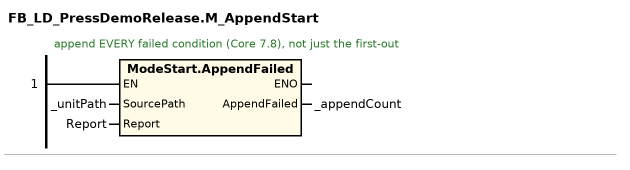
// NETWORK 1
// append EVERY failed condition (Core 7.8), not just the first-out
_appendCount := ModeStart.AppendFailed(SourcePath := _unitPath, Report := Report);
END_METHOD

// Deliberately ST, in a POU whose interlocks are ladder. This method is TARGET
// DISPATCH and bounded-report bookkeeping - matching a path against three child
// names and, failing that, writing five fields of one report row. None of that
// is condition logic, which is what O2's choice of language is about, and a
// ladder rendition of it would be longer, harder to read and no more
// demonstrative. Per-method language choice is exactly what TwinCAT offers.
METHOD M_AppendManual
VAR_INPUT
    TargetPath : STRING(255);
    Value : DINT;
    PressRam : REFERENCE TO FB_CylinderCM;
    Door : REFERENCE TO FB_CylinderCM;
    PartSlide : REFERENCE TO FB_CylinderCM;
END_VAR
VAR_IN_OUT
    Report : ST_ReleaseReport;
END_VAR
IF TargetPath = PressRam.Name THEN
    PressRam.AppendDirectionalRelease(Value := Value, Report := Report);
ELSIF TargetPath = Door.Name THEN
    Door.AppendDirectionalRelease(Value := Value, Report := Report);
ELSIF TargetPath = PartSlide.Name THEN
    PartSlide.AppendDirectionalRelease(Value := Value, Report := Report);
ELSE
    IF Report.Count < PL_Fraktal.MAX_RELEASE_REASONS THEN
        Report.Count := Report.Count + 1;
        Report.Reasons[Report.Count].Description := 'std.error.unsupportedManualTarget';
        Report.Reasons[Report.Count].ReasonCode := E_Reason.UNSUPPORTED_COMMAND;
        Report.Reasons[Report.Count].SourcePath := _unitPath;
        Report.Reasons[Report.Count].Kind := E_ReleaseKind.OTHER;
        Report.Reasons[Report.Count].Bypassable := FALSE;
    ELSE
        ; // bounded report is full; no array write is attempted
    END_IF
END_IF
END_METHOD

END_FUNCTION_BLOCK

// ---- PressTests/FB_FaultRecovery_Tests.TcPOU
// Regression suite for the press hard-lock: an AUTO cycle reached N200 (ram down),
// the operator released the two-hand button mid-stroke — the designed way to stop a
// stroke — and NO panel action could recover the machine.
//
// Measured on the live PLC, the lock was two latches deep:
//   1. the lost permissive was classified as a FAULT, so the only exit was
//      Reset -> IDLE, and the fault's own condition ("two-hand held during a
//      stroke") could only be re-established by starting;
//   2. OperatorReset skipped an ACTIVE event and left both Execute inputs asserted,
//      and §6.1's Execute-drop reset — the sole exit from a latched terminal state —
//      needs them low. A Unit that is not BUSY never calls _M_Dispatch again, so the
//      frozen step holding `PressRam.Execute := TRUE` could never clear it, and the
//      next HOME re-issued an already-TRUE input: no rising edge, ram stuck in its
//      latched state, Unit re-adopting the fault through the §8.2 rollup.
//
// The ram is held mid-stroke deterministically by NOT calling its sim plant, so its
// position feedback never arrives (MoveTimeout is T#2S and a TON cannot advance
// inside one PLC scan, so it cannot expire here and turn the wait into a timeout).
FUNCTION_BLOCK FB_FaultRecovery_Tests EXTENDS TcUnit.FB_TestSuite
VAR
    Press : FB_PressDemoUnit;
    PressHal, DoorHal, SlideHal : ST_CylinderHal;
    TwoHandHal : ST_TwoHandHal;
    PowerHal : ST_PowerGroupHal;
    PartPresentHal : ST_DigitalInputHal;
    AirPressureHal : ST_AirPressureHal;
    PressSim, DoorSim, SlideSim : FB_CylinderSim;
    Recipe : FB_LocalRecipeProvider;
    Cfg : ST_PneumaticPressParCfg;
    Domain : ST_ControlDomainStatus;
    Release : ST_ReleaseReport;
    Wired : BOOL;
    i : INT;
END_VAR

IF NOT Wired THEN
    // A non-zero dwell keeps N220 open for the dwell-hold assertions; a TON never
    // advances inside a scan, so the dwell simply does not elapse during a test.
    Cfg.PressSettleTime := T#500MS;
    Cfg.TransferSettleTime := T#0S;
    Cfg.IdealCycleMs := 1000;
    Cfg.BaselineWorkMs := 900;
    // RequireTwoHandStart is STATION config now (S3.8a), not recipe data. The
    // bench takes it from the Unit's own persistent image, which Setup
    // initializes to the fail-safe TRUE on a first boot - and which no recipe
    // can reach, which is exactly why it was moved.
    Recipe.Register(ModelCode := '', RecipeKey := 'PneumaticPressUnit', pData := ADR(Cfg), Size := SIZEOF(Cfg));
    PressHal.RetractedFb := TRUE; DoorHal.RetractedFb := TRUE; SlideHal.RetractedFb := TRUE;
    Press.Setup(Name := 'Test.Recovery', PressHal := PressHal, DoorHal := DoorHal,
        SlideHal := SlideHal, TwoHandHal := TwoHandHal, PowerHal := PowerHal,
        PartPresentHal := PartPresentHal, AirPressureHal := AirPressureHal, Recipe := Recipe);
    PressSim.Setup(HalRef := PressHal, TravelTime := T#0S);
    DoorSim.Setup(HalRef := DoorHal, TravelTime := T#0S);
    SlideSim.Setup(HalRef := SlideHal, TravelTime := T#0S);
    PowerHal.SafetyPermit := TRUE; PowerHal.FieldbusHealthy := TRUE; PowerHal.PowerFeedback := TRUE;
    TwoHandHal.FieldbusHealthy := TRUE;
    PartPresentHal.Quality := TRUE; PartPresentHal.Value := TRUE;
    AirPressureHal.Quality := TRUE;
    AirPressureHal.LowPressure := FALSE; AirPressureHal.OperatingPressure := TRUE;
    Domain.Present := TRUE; Domain.Id := 'TEST-RECOVERY'; Domain.ReadyForStart := TRUE;
    Domain.Safety.Present := TRUE; Domain.Safety.AllSafe := TRUE;
    Domain.ControlPower.Present := TRUE; Domain.ControlPower.ControlOn := TRUE;
    Press.ControlDomain := Domain;
    Press.SetMode(Mode := E_Mode.AUTO);
    Press();
    Wired := TRUE;
END_IF
Two_hand_release_mid_stroke_holds_the_ram();
Two_hand_release_in_the_dwell_holds_and_restores();
Air_loss_mid_stroke_holds_and_resumes();
Latched_fault_recovers_with_one_operator_reset();
Reset_never_bypasses_a_live_condition();

// Drive the fixture from the load-safe position to N200 with the ram commanded
// EXTEND and still travelling. The ram's plant model is deliberately NOT ticked, so
// its extended feedback never arrives and the stroke stays in progress.
METHOD PROTECTED _M_RunToRamDown : BOOL
VAR
    scan : INT;
END_VAR
TwoHandHal.LeftPressed := FALSE; TwoHandHal.RightPressed := FALSE;
TwoHandHal.SafeActive := FALSE;
Press();                                     // clear any stale start pulse
TwoHandHal.LeftPressed := TRUE; TwoHandHal.RightPressed := TRUE;
TwoHandHal.SafeActive := TRUE;               // physical start edge (§3.4.2, non-safety)
FOR scan := 1 TO 40 DO
    DoorSim(); SlideSim(); Press();
END_FOR
_M_RunToRamDown := _M_AtStep(StepNo := 200) AND Press.PressRam.Busy;
END_METHOD

// Drive the fixture to N180 with the door commanded EXTEND and still travelling.
// N180 AWAITS the door, so a door fault there is adopted by the Unit through the
// rollup (§8.2) - unlike N200, which owns the ram's failure itself. The door's
// plant model is deliberately NOT ticked, so its closed feedback never arrives.
METHOD PROTECTED _M_RunToDoorClosing : BOOL
VAR
    scan : INT;
END_VAR
TwoHandHal.LeftPressed := FALSE; TwoHandHal.RightPressed := FALSE;
TwoHandHal.SafeActive := FALSE;
Press();                                     // clear any stale start pulse
TwoHandHal.LeftPressed := TRUE; TwoHandHal.RightPressed := TRUE;
TwoHandHal.SafeActive := TRUE;               // physical start edge (§3.4.2, non-safety)
FOR scan := 1 TO 40 DO
    PressSim(); SlideSim(); Press();
    IF _M_AtStep(StepNo := 180) AND Press.Door.Busy THEN
        EXIT;
    END_IF
END_FOR
_M_RunToDoorClosing := _M_AtStep(StepNo := 180) AND Press.Door.Busy;
END_METHOD

// Leave the fixture where every test in this suite expects to find it: AUTO, stopped,
// no blocking event, ram/door/slide back at the load-safe position, two-hand released.
METHOD PROTECTED _M_ReturnToIdle
VAR
    scan : INT;
END_VAR
TwoHandHal.LeftPressed := FALSE; TwoHandHal.RightPressed := FALSE;
TwoHandHal.SafeActive := FALSE;
AirPressureHal.LowPressure := FALSE; AirPressureHal.OperatingPressure := TRUE;
DoorHal.ExtendedFb := FALSE;                 // undo a contradictory door position
Press.OperatorReset();
// HOME is interruptible and uses the normal immediate mode-exit handshake. This
// deterministically abandons an open AUTO dwell without pretending rapid calls
// advance its 500 ms TON.
Press.SetMode(Mode := E_Mode.HOME);
FOR scan := 1 TO 8 DO
    PressSim(); DoorSim(); SlideSim(); Press();
END_FOR
IF (Press.ModeActive = E_Mode.HOME) AND (Press.State = E_ExecState.READY) THEN
    Press.Start();
END_IF
FOR scan := 1 TO 30 DO
    PressSim(); DoorSim(); SlideSim(); Press();
END_FOR
Press.Stop();
FOR scan := 1 TO 4 DO
    PressSim(); DoorSim(); SlideSim(); Press();
END_FOR
Press.SetMode(Mode := E_Mode.AUTO);
FOR scan := 1 TO 6 DO
    PressSim(); DoorSim(); SlideSim(); Press();
END_FOR
END_METHOD

// Defect B: releasing the button mid-stroke is expected operator behaviour, so it
// belongs in HELD (suspend, resume when restored), not in a fault whose only exit is
// Reset -> IDLE. Nothing is relaxed: the output is still withheld by the same permit.
METHOD Two_hand_release_mid_stroke_holds_the_ram
TEST('Two_hand_release_mid_stroke_holds_the_ram');
AssertTrue(Condition := _M_RunToRamDown(),
    Message := 'fixture reaches N200 with the ram travelling');
AssertTrue(Condition := PressHal.ExtendOut, Message := 'ram is driving down');

// The operator lets go, mid-stroke.
TwoHandHal.LeftPressed := FALSE; TwoHandHal.RightPressed := FALSE;
TwoHandHal.SafeActive := FALSE;
DoorSim(); SlideSim(); Press();
DoorSim(); SlideSim(); Press();

AssertFalse(Condition := PressHal.ExtendOut,
    Message := 'the permit still withholds the output — the interlock is untouched');
AssertTrue(Condition := Press.PressRam.Held, Message := 'ram is HELD (§6.1)');
AssertFalse(Condition := Press.PressRam.Error, Message := 'a released two-hand is not a ram fault');
AssertFalse(Condition := Press.Error, Message := 'and it is not a Unit fault either');
AssertFalse(Condition := Press.AlarmLog.Blocking,
    Message := 'no MANUAL_RESET event, so nothing blocks the restart (§8.3(b))');
AssertTrue(Condition := Press.Held, Message := 'the Unit reports the awaited hold (§8.2)');
AssertEquals_STRING(Expected := 'project.interlock.pressRequiresTwoHandHeld',
    Actual := Press.Status.Diagnostic.Description,
    Message := 'the operator sees WHICH condition is missing, not a composite key (§6.9)');
AssertEquals_STRING(Expected := 'Test.Recovery.PressRam',
    Actual := Press.Status.Diagnostic.SourcePath,
    Message := 'the held module names itself, not the Unit');

// Pressing again resumes the same stroke — no reset, no restart, no lost part.
TwoHandHal.LeftPressed := TRUE; TwoHandHal.RightPressed := TRUE;
TwoHandHal.SafeActive := TRUE;
DoorSim(); SlideSim(); Press();
DoorSim(); SlideSim(); Press();
AssertTrue(Condition := PressHal.ExtendOut, Message := 'resume re-energizes the ram');
AssertFalse(Condition := Press.PressRam.Held, Message := 'hold clears itself when the button returns');
FOR i := 1 TO 6 DO
    PressSim(); DoorSim(); SlideSim(); Press();      // let the stroke finish now
END_FOR
AssertTrue(Condition := _M_AtStep(StepNo := 220),
    Message := 'the suspended stroke completes and the cycle carries on');
_M_ReturnToIdle();
TEST_FINISHED();
END_METHOD

// N220 holds the press force through the dwell. The force is the valve latched by the
// EXTEND that N200 already completed, so a withdraw needs an explicit restore — the
// case a hold at the CM alone does not cover.
METHOD Two_hand_release_in_the_dwell_holds_and_restores
TEST('Two_hand_release_in_the_dwell_holds_and_restores');
AssertTrue(Condition := _M_RunToRamDown(), Message := 'fixture reaches N200');
FOR i := 1 TO 6 DO
    PressSim(); DoorSim(); SlideSim(); Press();      // complete the stroke -> dwell
END_FOR
AssertTrue(Condition := _M_AtStep(StepNo := 220), Message := 'dwelling at N220');
AssertTrue(Condition := PressHal.ExtendOut, Message := 'press force is applied during the dwell');

TwoHandHal.LeftPressed := FALSE; TwoHandHal.RightPressed := FALSE;
TwoHandHal.SafeActive := FALSE;
PressSim(); DoorSim(); SlideSim(); Press();
AssertFalse(Condition := PressHal.ExtendOut, Message := 'releasing the button stops pressing');
AssertFalse(Condition := Press.Error, Message := 'and does not fault the cycle');
AssertTrue(Condition := _M_AtStep(StepNo := 220), Message := 'the dwell holds where it was');
AssertFalse(Condition := Press.CurrentStep.Conds[1].Ok,
    Message := 'the named dwell condition shows FALSE (§6.9(b))');
AssertEquals_STRING(Expected := 'project.condition.twoHandHeldDuringPress',
    Actual := Press.CurrentStep.Conds[1].Label,
    Message := 'the recorded wait names the dwell permit');

TwoHandHal.LeftPressed := TRUE; TwoHandHal.RightPressed := TRUE;
TwoHandHal.SafeActive := TRUE;
PressSim(); DoorSim(); SlideSim(); Press();
PressSim(); DoorSim(); SlideSim(); Press();
AssertTrue(Condition := PressHal.ExtendOut,
    Message := 'pressing again restores the press force (RestoreOutputs)');
_M_ReturnToIdle();
TEST_FINISHED();
END_METHOD

// Air is restored by the process, not repaired, so losing it mid-stroke is HELD
// (§6.1): the ram's own process condition withdraws its valve, the Unit reports the
// hold by name, nothing is latched, and the stroke resumes when pressure returns.
METHOD Air_loss_mid_stroke_holds_and_resumes
TEST('Air_loss_mid_stroke_holds_and_resumes');
AssertTrue(Condition := _M_RunToRamDown(), Message := 'fixture reaches N200');
AssertTrue(Condition := PressHal.ExtendOut, Message := 'ram is driving down');
AirPressureHal.OperatingPressure := FALSE;
AirPressureHal.LowPressure := TRUE;
FOR i := 1 TO 3 DO
    DoorSim(); SlideSim(); Press();
END_FOR
AssertFalse(Condition := PressHal.ExtendOut, Message := 'the ram valve is withdrawn');
AssertTrue(Condition := Press.PressRam.Held, Message := 'the ram is HELD, not faulted');
AssertFalse(Condition := Press.Error, Message := 'the Unit does not fault');
AssertFalse(Condition := Press.AlarmLog.Blocking, Message := 'and nothing needs a reset');
AssertTrue(Condition := Press.Held, Message := 'the Unit reports the hold');
AssertEquals_STRING(Expected := 'project.interlock.pressRequiresAirPressure',
    Actual := Press.Status.Diagnostic.Description,
    Message := 'by the missing condition, not a composite key (§6.9)');
AirPressureHal.OperatingPressure := TRUE;
AirPressureHal.LowPressure := FALSE;
FOR i := 1 TO 3 DO
    DoorSim(); SlideSim(); Press();
END_FOR
AssertTrue(Condition := PressHal.ExtendOut, Message := 'pressure back: the stroke resumes by itself');
AssertFalse(Condition := Press.PressRam.Held, Message := 'and the hold has cleared');
_M_ReturnToIdle();
TEST_FINISHED();
END_METHOD

// Defect A + C, the actual hard-lock: a genuine fault while the ram is travelling
// left a state the press could not get out of. ONE reset has to make HOME runnable
// again. The fault is a contradictory door position (both end sensors) while the
// door closes - a defect, unlike air loss, which the process restores and which
// therefore holds (Air_loss_mid_stroke_holds_and_resumes).
METHOD Latched_fault_recovers_with_one_operator_reset
TEST('Latched_fault_recovers_with_one_operator_reset');
AssertTrue(Condition := _M_RunToDoorClosing(), Message := 'fixture reaches N180 with the door closing');

// Both door end sensors while it closes: CYL_BOTH_SENSORS. N180 awaits the door, so
// the Unit adopts it with the chain frozen where it had asserted Door.Execute.
DoorHal.ExtendedFb := TRUE;
FOR i := 1 TO 3 DO
    PressSim(); SlideSim(); Press();
END_FOR

AssertTrue(Condition := Press.Error, Message := 'a contradictory door position is a real fault');
AssertTrue(Condition := Press.AlarmLog.Blocking, Message := 'and raises a blocking event (§8.3(b))');
AssertEquals_DINT(Expected := TO_DINT(E_AlarmState.ACTIVE),
    Actual := TO_DINT(Press.AlarmLog.Active[1].State),
    Message := 'the event is ACTIVE — it never reached WAIT_RESET');
// The two latches that made this unrecoverable:
AssertTrue(Condition := Press.Execute, Message := 'the run command is still asserted');
AssertTrue(Condition := Press.Door.Execute,
    Message := 'and so is the child command the frozen chain issued');

// Correct the sensor: the CAUSE is gone, but the latched state is not, and Start stays shut.
DoorHal.ExtendedFb := FALSE;
PressSim(); SlideSim(); Press();
Press.ReleaseReportStart(Report := Release);
AssertFalse(Condition := Release.Released,
    Message := 'a cleared cause does not by itself unlatch the Unit');

// ONE operator action.
AssertTrue(Condition := Press.OperatorReset(), Message := 'the reset is accepted');
AssertFalse(Condition := Press.AlarmLog.Blocking,
    Message := 'an ACTIVE MANUAL_RESET event closes on a deliberate reset (§8.3(b))');
AssertEquals_DINT(Expected := TO_DINT(E_AlarmState.CLOSED),
    Actual := TO_DINT(Press.AlarmLog.Active[1].State), Message := 'slot released');
// Guarded: an unguarded Ring[RingHead] with nothing closed reads index 0 and
// page-faults the runtime, taking every later test down with this one.
IF Press.AlarmLog.RingHead > 0 THEN
    AssertTrue(Condition := Press.AlarmLog.Ring[Press.AlarmLog.RingHead].Duration >= T#0S,
        Message := 'the closed event still carries a Duration (§8.3(a))');
ELSE
    AssertTrue(Condition := FALSE, Message := 'the reset closed an event into the ring');
END_IF
AssertFalse(Condition := Press.Execute, Message := 'the stale run command is released');
AssertFalse(Condition := Press.Door.Execute, Message := 'the stranded child command is released');

DoorSim(); SlideSim(); Press();
DoorSim(); SlideSim(); Press();
AssertTrue(Condition := Press.State = E_ExecState.READY,
    Message := 'the Unit is READY after the inherited Execute-drop reset (§6.1)');
AssertTrue(Condition := Press.Door.State = E_ExecState.READY,
    Message := 'and so is the door, so it can take a fresh command edge');

// Defect C: the recovery sequence is now reachable, under normal access authority.
AssertTrue(Condition := Press.SetMode(Mode := E_Mode.HOME), Message := 'HOME can be selected');
Press();
AssertTrue(Condition := Press.Start(), Message := 'HOME starts with no further operator action');
FOR i := 1 TO 30 DO
    PressSim(); DoorSim(); SlideSim(); Press();
END_FOR
AssertTrue(Condition := Press.OutImm.Homed, Message := 'HOME reaches the load-safe position');
_M_ReturnToIdle();
TEST_FINISHED();
END_METHOD

// The reset closes a latched event even while a start condition is unsatisfied, which
// is only safe because it clears the LATCH and never the condition. Proof: fault the
// Unit, take the air away, reset, then watch the release report keep Start shut on
// that live condition.
METHOD Reset_never_bypasses_a_live_condition
TEST('Reset_never_bypasses_a_live_condition');
AssertTrue(Condition := _M_RunToDoorClosing(), Message := 'fixture reaches N180 with the door closing');
DoorHal.ExtendedFb := TRUE;
FOR i := 1 TO 3 DO
    PressSim(); SlideSim(); Press();
END_FOR
AssertTrue(Condition := Press.AlarmLog.Blocking, Message := 'faulted on the contradictory door position');
DoorHal.ExtendedFb := FALSE;
AirPressureHal.OperatingPressure := FALSE;
AirPressureHal.LowPressure := TRUE;
PressSim(); SlideSim(); Press();

AssertTrue(Condition := Press.OperatorReset(), Message := 'reset is accepted with the cause still live');
DoorSim(); SlideSim(); Press();
AssertFalse(Condition := Press.AlarmLog.Blocking, Message := 'the latch is cleared');
Press.ReleaseReportStart(Report := Release);
AssertFalse(Condition := Release.Released,
    Message := 'but Start is still refused — the reset cleared the latch, not the condition');
AssertFalse(Condition := Press.ReleaseConditions.ModeStartAirPressureOk,
    Message := 'and the live condition is still reported by name (§7.8)');
AssertFalse(Condition := PressHal.ExtendOut,
    Message := 'no output is restored by a reset');
_M_ReturnToIdle();
TEST_FINISHED();
END_METHOD

METHOD PRIVATE _M_AtStep : BOOL
VAR_INPUT
    StepNo : INT;
END_VAR
VAR
    branchIndex : INT;
    rowIndex : INT;
END_VAR
// CurrentStep is main-line only. SFC's ram leg has its own §3.13 cursor.
_M_AtStep := FALSE;
FOR branchIndex := 0 TO PL_Fraktal.MAX_PARALLEL_BRANCHES DO
    rowIndex := Press.ActiveSteps[branchIndex].RowIdx;
    IF (rowIndex >= 1) AND (rowIndex <= Press.SequenceStepCount) THEN
        IF Press.SequenceStepDef[rowIndex].StepNo = StepNo THEN
            _M_AtStep := TRUE;
            RETURN;
        END_IF
    END_IF
END_FOR
END_METHOD

END_FUNCTION_BLOCK

// ---- Fraktal_Press_Demo/01_PneumaticPress/Recipes/FB_PressRecipeCatalog.TcPOU
// Owner-local recipe engineering data: model identities and their typed Unit records.
// Generic validation/storage remains in FB_LocalRecipeProvider; process behavior
// remains in the project-owned FB_PressDemoUnit. MAIN only composes the two.
FUNCTION_BLOCK FB_PressRecipeCatalog
VAR_OUTPUT
    {attribute 'OPC.UA.DA' := '0'}
    Provider : FB_LocalRecipeProvider;
END_VAR
VAR PERSISTENT
    // §3.8b - the records are edited through the Unit's model data (any model;
    // the provider's Save writes here) and must outlive a restart, so they are
    // retained and seeded only once.
    _default : ST_PneumaticPressParCfg;
    _aluminum : ST_PneumaticPressParCfg;
    _plastic : ST_PneumaticPressParCfg;
    _steel : ST_PneumaticPressParCfg;
    _seeded : UINT;               // RECIPE_SEED once the defaults below were written
END_VAR
VAR
    _model : ST_ModelId;
    _configured : BOOL;
END_VAR
VAR CONSTANT
    // Bump to re-seed every record with the design values below (a download that
    // changes them, or a record layout change).
    RECIPE_SEED : UINT := 1;
END_VAR

// Static catalog: no cyclic work.

METHOD Setup : BOOL
VAR_INPUT
    UnitRef : REFERENCE TO FB_PressDemoUnit;
END_VAR
VAR
    Ok : BOOL;
END_VAR
IF _configured THEN
    Setup := TRUE;
    RETURN;
END_IF

// §8.11 per-model performance references: IdealCycleMs feeds OEE Performance
// (§8.5.1); BaselineWorkMs arms the WORK-time degradation watch (§8.11.4(d)).
// Values = design cycle for this training cell (motions + settle + dwell).
// Seeded once: afterwards the retained records hold what was edited.
IF _seeded <> RECIPE_SEED THEN
    _default.PressSettleTime := T#500MS;
    _default.TransferSettleTime := T#100MS;
    _default.IdealCycleMs := 6000;
    _default.BaselineWorkMs := 6000;
    _aluminum.PressSettleTime := T#300MS;
    _aluminum.TransferSettleTime := T#80MS;
    _aluminum.IdealCycleMs := 5700;
    _aluminum.BaselineWorkMs := 5700;
    _plastic.PressSettleTime := T#650MS;
    _plastic.TransferSettleTime := T#120MS;
    _plastic.IdealCycleMs := 6200;
    _plastic.BaselineWorkMs := 6200;
    _steel.PressSettleTime := T#1200MS;
    _steel.TransferSettleTime := T#150MS;
    _steel.IdealCycleMs := 6800;
    _steel.BaselineWorkMs := 6800;
    _seeded := RECIPE_SEED;
END_IF

Ok := Provider.Register(ModelCode := '', RecipeKey := 'PneumaticPressUnit',
    pData := ADR(_default), Size := SIZEOF(_default));
Ok := Provider.Register(ModelCode := 'ALUMINUM', RecipeKey := 'PneumaticPressUnit',
    pData := ADR(_aluminum), Size := SIZEOF(_aluminum)) AND Ok;
Ok := Provider.Register(ModelCode := 'PLASTIC', RecipeKey := 'PneumaticPressUnit',
    pData := ADR(_plastic), Size := SIZEOF(_plastic)) AND Ok;
Ok := Provider.Register(ModelCode := 'STEEL', RecipeKey := 'PneumaticPressUnit',
    pData := ADR(_steel), Size := SIZEOF(_steel)) AND Ok;

_model.ModelCode := 'ALUMINUM';
Ok := UnitRef.RegisterAvailableModel(Id := _model) AND Ok;
_model.ModelCode := 'PLASTIC';
Ok := UnitRef.RegisterAvailableModel(Id := _model) AND Ok;
_model.ModelCode := 'STEEL';
Ok := UnitRef.RegisterAvailableModel(Id := _model) AND Ok;

_configured := Ok;
Setup := Ok;
END_METHOD

END_FUNCTION_BLOCK
